// TwinCAT 3 PLC project Untitled1
// ProgramVersion: 3.1.4026.14
// libraries:
//   Tc2_EtherCAT, * (Beckhoff Automation GmbH)
//   Tc2_MC2, * (Beckhoff Automation GmbH)
//   Tc2_Standard, * (Beckhoff Automation GmbH)
//   Tc2_System, * (Beckhoff Automation GmbH)
//   Tc2_Utilities, * (Beckhoff Automation GmbH)
//   Tc3_Module, * (Beckhoff Automation GmbH)
// project tree:
//   DUTs/ ENUM_HardwareCheckState.TcDUT, ENUM_LinearActuatorState.TcDUT, ENUM_StepperMotorState.TcDUT, ST_AlarmEntry.TcDUT, ST_LinearActuator.TcDUT, ST_Alarm.TcDUT, ST_LinearActuatorCommand.TcDUT, ST_LinearTable.TcDUT, ST_LookupEntry.TcDUT, ST_StepperMotorCommand.TcDUT, ST_SystemAlarmStatus.TcDUT, ST_ZoneAlarmStatus.TcDUT
//   GVLs/ GVL_Alarms.TcGVL, GVL.TcGVL, GVL_CellPositionSensors.TcGVL, GVL_Steppers.TcGVL, GVL_LinearActuatorDriveControls.TcGVL, GVL_LinearActuatorProxSensors.TcGVL, GVL_LinearActuators.TcGVL, GVL_LinearActuatorRelays.TcGVL, GVL_Process.TcGVL, GVL_StepperPositions.TcGVL
//   / Main_Task.TcTTO
//   POUs/FunctionBlocks/ FB_AlarmStatusManager.TcPOU, FB_LinearActuator.TcPOU, FB_StepperMotor.TcPOU
//   POUs/Helper/ F_IssueActuatorCommand.TcPOU, F_GetLinearCommandMember.TcPOU, F_GetLinearCommandValue.TcPOU, F_GetStepperCommandMember.TcPOU, F_GetStepperCommandValue.TcPOU, F_GetStepperAlarmCondition.TcPOU, F_ValidateCommand.TcPOU, F_GetLinearActuatorAlarmCondition.TcPOU, F_GetMC2ErrorDescription.TcPOU
//   POUs/Programs/ PRG_AlarmHandler.TcPOU, PRG_CommandHandler.TcPOU, PRG_Cycle.TcPOU
// real-time tasks:
//   TASK Main_Task: cycle T#10ms, priority 1, ADS port 351
// motion (NC):
//   TASK NC-Task 1 SAF: cycle T#2ms, priority 4, ADS port 501
//   TASK NC-Task 1 SVB: cycle T#10ms, priority 12, ADS port 511
//   AXIS Stepper1 (id 1)
//     Dynamic: Acceleration=100, Deceleration=100, Jerk=66.6667
//     Velo: Maximum=150
//     OtherSettings: AllowMotionCmdToSlave=true
//     encoder EncType=19
//       EncPara: ScaleFactorNumerator=0.000115, MaxCount=#xffffffff
//         Inc: RefSoftSyncMask=#x0000ffff
//     drive DrvType=16
//       DrvPara: MaxCount=#xffffffff, DriveControlDWord=#x00020100
//         Analog: TorqueSetpointScale=10, ScaleFactorActTorque=0.1
//         TimeComp: TaskDelayCycles=1
//     controller CtrType=1
//       CtrPara: PriorControlFactor=1
//         Observer: BandWidth=20
//   AXIS Stepper2 (id 2)
//     Dynamic: Acceleration=99.9997, Deceleration=99.9997, Jerk=66.6667
//     Velo: Maximum=150
//     OtherSettings: AllowMotionCmdToSlave=true
//     encoder EncType=19
//       EncPara: MaxCount=#xffffffff
//         Inc: RefSoftSyncMask=#x0000ffff
//     drive DrvType=16
//       DrvPara: MaxCount=#xffffffff, DriveControlDWord=#x00020100
//         Analog: TorqueSetpointScale=10, ScaleFactorActTorque=0.1
//         TimeComp: TaskDelayCycles=1
//     controller CtrType=1
//       CtrPara: PriorControlFactor=1
//         Observer: BandWidth=20
//   AXIS Stepper3 (id 3)
//     Dynamic: Acceleration=100, Deceleration=100, Jerk=66.6667
//     Velo: Maximum=150
//     OtherSettings: AllowMotionCmdToSlave=true
//     encoder EncType=19
//       EncPara: MaxCount=#xffffffff
//         Inc: RefSoftSyncMask=#x0000ffff
//     drive DrvType=16
//       DrvPara: MaxCount=#xffffffff, DriveControlDWord=#x00020100
//         Analog: TorqueSetpointScale=10, ScaleFactorActTorque=0.1
//         TimeComp: TaskDelayCycles=1
//     controller CtrType=1
//       CtrPara: PriorControlFactor=1
//         Observer: BandWidth=20
//   AXIS Stepper4 (id 4)
//     Dynamic: Acceleration=100, Deceleration=100, Jerk=66.6667
//     Velo: Maximum=150
//     OtherSettings: AllowMotionCmdToSlave=true
//     encoder EncType=19
//       EncPara: MaxCount=#xffffffff
//         Inc: RefSoftSyncMask=#x0000ffff
//     drive DrvType=16
//       DrvPara: MaxCount=#xffffffff, DriveControlDWord=#x00020100
//         Analog: TorqueSetpointScale=10, ScaleFactorActTorque=0.1
//         TimeComp: TaskDelayCycles=1
//     controller CtrType=1
//       CtrPara: PriorControlFactor=1
//         Observer: BandWidth=20
// I/O:
//   DEVICE Périphérique 2 (EtherCAT) (disabled), AmsNetId 192.168.0.14.3.1
//     Terme 11 (EK1100) [EK1100 EtherCAT Coupler (2A E-Bus)]
//       Drive Stepper1 (EL7047) [EL7047 1Ch. Stepper motor output stage (50V, 5A)]
//       Drive Stepper2 (EL7047) [EL7047 1Ch. Stepper motor output stage (50V, 5A)]
//       Drive Stepper3 (EL7047) [EL7047 1Ch. Stepper motor output stage (50V, 5A)]
//       Drive Stepper4 (El7047) [EL7047 1Ch. Stepper motor output stage (50V, 5A)]
//   DEVICE Device 4 (EtherCAT) (disabled), AmsNetId 192.168.0.14.5.1
//     ECAT E-Bus (EK1200) [EK1200-5000 EtherCAT Power supply (2A E-Bus)]
//       Carte DO #1 (EL2809) [EL2809 16Ch. Dig. Output 24V, 0.5A]
//       Carte DO #2 (EL2809) [EL2809 16Ch. Dig. Output 24V, 0.5A]
//       Carte DO #3 (EL2809) [EL2809 16Ch. Dig. Output 24V, 0.5A]
//       Drive Stepper Rail1/2 (EL7062) [EL7062-0000 2Ch. Stepper motor output stage (48V, 3A)]
//       Drive Stepper Rail3/4 (EL7062) [EL7062-0000 2Ch. Stepper motor output stage (48V, 3A)]
//       E-Bus (EL9410) [EL9410 E-Bus Power Supplier  (Diagnostics)]
//       Carte DI #1 (EL1409) [EL1409 16Ch. Dig. Input 24V, 3ms]
//       Carte DI #2 (EL1409) [EL1409 16Ch. Dig. Input 24V, 3ms]
//       Carte DI #3 (EL1409) [EL1409 16Ch. Dig. Input 24V, 3ms]
//       Term 10 (EL4074) [EL4074 4K. Ana. Ausgang, +/-10V, +/-20mA, 16 Bit]
//       Term 8 (EL3078) [EL3078 8K. Ana. Eingang  +/-10V, +/-20mA]
//       Term 9 (EL3078) [EL3078 8K. Ana. Eingang  +/-10V, +/-20mA]
//       Carte Temperature Sensors #1 (EL3208-0010) [EL3208-0010 8Ch. Ana. Input PT1000 (RTD)]
//       Carte Temperature Sensors #2 (EL3208-0010) [EL3208-0010 8Ch. Ana. Input PT1000 (RTD)]
//       Carte Temperature Sensors #3 (EL3208-0010) [EL3208-0010 8Ch. Ana. Input PT1000 (RTD)]
//       End Terminal (EL9011) [EL9011 End Terminal]
// variable links:
//   NC-Task 1 SAF/Axes/Stepper1 <-> Device 4 (EtherCAT)/ECAT E-Bus (EK1200)/Drive Stepper Rail1/2 (EL7062)
//     Drive/Inputs/In/nDataIn1 <-> DRV Following error actual value Channel 1/Following error actual value
//     Drive/Inputs/In/nDcOutputTime <-> InfoData/DcOutputShift
//     Drive/Inputs/In/nState1 <-> DRV Statusword Channel 1/Statusword
//     Drive/Inputs/In/nState2 <-> DRV Statusword Channel 1/Statusword @bit 8
//     Drive/Inputs/In/nState4 @bit 1 <-> WcState/InputToggle
//     Drive/Inputs/In/nState4 <-> WcState/WcState
//     Drive/Outputs/Out/nCtrl1 <-> DRV Controlword Channel 1/Controlword
//     Drive/Outputs/Out/nCtrl2 <-> DRV Controlword Channel 1/Controlword @bit 8
//     Drive/Outputs/Out/nDataOut1 <-> DRV Target position Channel 1/Target position
//     Enc/Inputs/In/nDataIn1 <-> FB Position Channel 1/Position
//     Enc/Inputs/In/nDcInputTime <-> InfoData/DcInputShift
//     Enc/Inputs/In/nState4 @bit 1 <-> WcState/InputToggle
//     Enc/Inputs/In/nState4 <-> WcState/WcState
//   NC-Task 1 SAF/Axes/Stepper2 <-> Device 4 (EtherCAT)/ECAT E-Bus (EK1200)/Drive Stepper Rail1/2 (EL7062)
//     Drive/Inputs/In/nDataIn1 <-> DRV Following error actual value Channel 2/Following error actual value
//     Drive/Inputs/In/nDcOutputTime <-> InfoData/DcOutputShift
//     Drive/Inputs/In/nState1 <-> DRV Statusword Channel 2/Statusword
//     Drive/Inputs/In/nState2 <-> DRV Statusword Channel 2/Statusword @bit 8
//     Drive/Inputs/In/nState4 @bit 1 <-> WcState/InputToggle
//     Drive/Inputs/In/nState4 <-> WcState/WcState
//     Drive/Outputs/Out/nCtrl1 <-> DRV Controlword Channel 2/Controlword
//     Drive/Outputs/Out/nCtrl2 <-> DRV Controlword Channel 2/Controlword @bit 8
//     Drive/Outputs/Out/nDataOut1 <-> DRV Target position Channel 2/Target position
//     Enc/Inputs/In/nDataIn1 <-> FB Position Channel 2/Position
//     Enc/Inputs/In/nDcInputTime <-> InfoData/DcInputShift
//     Enc/Inputs/In/nState4 @bit 1 <-> WcState/InputToggle
//     Enc/Inputs/In/nState4 <-> WcState/WcState
//   NC-Task 1 SAF/Axes/Stepper3 <-> Device 4 (EtherCAT)/ECAT E-Bus (EK1200)/Drive Stepper Rail3/4 (EL7062)
//     Drive/Inputs/In/nDataIn1 <-> DRV Following error actual value Channel 1/Following error actual value
//     Drive/Inputs/In/nDcOutputTime <-> InfoData/DcOutputShift
//     Drive/Inputs/In/nState1 <-> DRV Statusword Channel 1/Statusword
//     Drive/Inputs/In/nState2 <-> DRV Statusword Channel 1/Statusword @bit 8
//     Drive/Inputs/In/nState4 @bit 1 <-> WcState/InputToggle
//     Drive/Inputs/In/nState4 <-> WcState/WcState
//     Drive/Outputs/Out/nCtrl1 <-> DRV Controlword Channel 1/Controlword
//     Drive/Outputs/Out/nCtrl2 <-> DRV Controlword Channel 1/Controlword @bit 8
//     Drive/Outputs/Out/nDataOut1 <-> DRV Target position Channel 1/Target position
//     Enc/Inputs/In/nDataIn1 <-> FB Position Channel 1/Position
//     Enc/Inputs/In/nDcInputTime <-> InfoData/DcInputShift
//     Enc/Inputs/In/nState4 @bit 1 <-> WcState/InputToggle
//     Enc/Inputs/In/nState4 <-> WcState/WcState
//   NC-Task 1 SAF/Axes/Stepper4 <-> Device 4 (EtherCAT)/ECAT E-Bus (EK1200)/Drive Stepper Rail3/4 (EL7062)
//     Drive/Inputs/In/nDataIn1 <-> DRV Following error actual value Channel 2/Following error actual value
//     Drive/Inputs/In/nDcOutputTime <-> InfoData/DcOutputShift
//     Drive/Inputs/In/nState1 <-> DRV Statusword Channel 2/Statusword
//     Drive/Inputs/In/nState2 <-> DRV Statusword Channel 2/Statusword @bit 8
//     Drive/Inputs/In/nState4 @bit 1 <-> WcState/InputToggle
//     Drive/Inputs/In/nState4 <-> WcState/WcState
//     Drive/Outputs/Out/nCtrl1 <-> DRV Controlword Channel 2/Controlword
//     Drive/Outputs/Out/nCtrl2 <-> DRV Controlword Channel 2/Controlword @bit 8
//     Drive/Outputs/Out/nDataOut1 <-> DRV Target position Channel 2/Target position
//     Enc/Inputs/In/nDataIn1 <-> FB Position Channel 2/Position
//     Enc/Inputs/In/nDcInputTime <-> InfoData/DcInputShift
//     Enc/Inputs/In/nState4 @bit 1 <-> WcState/InputToggle
//     Enc/Inputs/In/nState4 <-> WcState/WcState
//   Untitled1/Untitled1 Instance <-> Device 4 (EtherCAT)/ECAT E-Bus (EK1200)/Carte DI #1 (EL1409)
//     Main_Task Inputs/GVL_CellPositionSensors.Cell_Pos{1..6} <-> DIP Inputs/Cell Position {1..6}  (6 links)
//     Main_Task Inputs/GVL_LinearActuatorProxSensors.Tri{1..4}_Prox_In <-> DIP Inputs/Triangle Rétractable Chariot{1..4} Prox In  (4 links)
//     Main_Task Inputs/GVL_LinearActuatorProxSensors.Tri{1..4}_Prox_Out <-> DIP Inputs/Triangle Rétractable Chariot{1..4} Prox Out  (4 links)
//   Untitled1/Untitled1 Instance <-> Device 4 (EtherCAT)/ECAT E-Bus (EK1200)/Carte DI #2 (EL1409)
//     Main_Task Inputs/GVL_LinearActuatorProxSensors.Gui1_Prox_In_Slow <-> DIP Inputs/Gui1 Prox In Slow
//     Main_Task Inputs/GVL_LinearActuatorProxSensors.Gui2_Prox_In_Slow <-> DIP Inputs/Gui2 Prox In Slow
//     Main_Task Inputs/GVL_LinearActuatorProxSensors.Gui1_Prox_Out <-> DIP Inputs/Gui1 Prox Out
//     Main_Task Inputs/GVL_LinearActuatorProxSensors.Gui2_Prox_Out <-> DIP Inputs/Gui2 Prox Out
//     Main_Task Inputs/GVL_LinearActuatorProxSensors.Gui1_Prox_Out_Slow <-> DIP Inputs/Gui1 Prox Out Slow
//     Main_Task Inputs/GVL_LinearActuatorProxSensors.Gui2_Prox_Out_Slow <-> DIP Inputs/Gui2 Prox Out Slow
//     Main_Task Inputs/GVL_Steppers.Rail1_Prox <-> DIP Inputs/Prox Homing Rail1
//     Main_Task Inputs/GVL_Steppers.Rail2_Prox <-> DIP Inputs/Prox Homing Rail2
//   Untitled1/Untitled1 Instance <-> Device 4 (EtherCAT)/ECAT E-Bus (EK1200)/Carte DI #3 (EL1409)
//     Main_Task Inputs/GVL.PLC_Fan_Steppers <-> DIP Inputs/Fan Stepper Status
//     Main_Task Inputs/GVL.ResetSafety <-> DIP Inputs/Reset Safety
//     Main_Task Inputs/GVL.SafetyRelayStatus <-> DIP Inputs/Safety Relay Status
//     Main_Task Inputs/GVL.StartCycle <-> DIP Inputs/Start Cycle
//     Main_Task Inputs/GVL.StopCycle <-> DIP Inputs/Stop Cycle
//     Main_Task Inputs/GVL_LinearActuatorDriveControls.Cmp1_Mot_Fault <-> DIP Inputs/Cmp1 Fault
//     Main_Task Inputs/GVL_LinearActuatorDriveControls.Cmp2_Mot_Fault <-> DIP Inputs/Cmp2 Fault
//     Main_Task Inputs/GVL_LinearActuatorDriveControls.Gui1_Mot_Fault <-> DIP Inputs/Gui1 Fault
//     Main_Task Inputs/GVL_LinearActuatorDriveControls.Gui2_Mot_Fault <-> DIP Inputs/Gui2 Fault
//     Main_Task Inputs/GVL_LinearActuatorProxSensors.Piv1_Prox_In <-> DIP Inputs/Piv1 Prox In
//     Main_Task Inputs/GVL_LinearActuatorProxSensors.Piv1_Prox_Out <-> DIP Inputs/Piv1 Prox Out
//     Main_Task Inputs/GVL_Steppers.Rail3_Prox <-> DIP Inputs/Prox Homing Rail3
//     Main_Task Inputs/GVL_Steppers.Rail4_Prox <-> DIP Inputs/Prox Homing Rail4
//   Untitled1/Untitled1 Instance <-> Device 4 (EtherCAT)/ECAT E-Bus (EK1200)/Carte DO #2 (EL2809)
//     Main_Task Outputs/GVL_LinearActuatorRelays.Piv1_Mot_Bw <-> Channel 13/Piv1 Backward
//     Main_Task Outputs/GVL_LinearActuatorRelays.Piv1_Mot_Fw <-> Channel 5/Piv1 Forward
//     Main_Task Outputs/GVL_LinearActuatorRelays.Tri1_Mot_Bw <-> Channel 1/Tri1 Pop-Up Forward
//     Main_Task Outputs/GVL_LinearActuatorRelays.Tri1_Mot_Fw <-> Channel 9/Tri1 Pop-Up Backward
//     Main_Task Outputs/GVL_LinearActuatorRelays.Tri2_Mot_Bw <-> Channel 11/Tri2 Pop-Up Backward
//     Main_Task Outputs/GVL_LinearActuatorRelays.Tri3_Mot_Bw <-> Channel 12/Tri3 Pop-Up Backward
//     Main_Task Outputs/GVL_LinearActuatorRelays.Tri4_Mot_Bw <-> Channel 10/Tri4 Pop-Up Backward
//     Main_Task Outputs/GVL_LinearActuatorRelays.Tri2_Mot_Fw <-> Channel 3/Tri2 Pop-Up Forward
//     Main_Task Outputs/GVL_LinearActuatorRelays.Tri3_Mot_Fw <-> Channel 4/Tri3 Pop-Up Forward
//     Main_Task Outputs/GVL_LinearActuatorRelays.Tri4_Mot_Fw <-> Channel 2/Tri4 Forward
//   Untitled1/Untitled1 Instance <-> Device 4 (EtherCAT)/ECAT E-Bus (EK1200)/Carte DO #3 (EL2809)
//     Main_Task Outputs/GVL_LinearActuatorDriveControls.Cmp1_Mot_Speed2 <-> Channel 4/Cmp1 Speed2
//     Main_Task Outputs/GVL_LinearActuatorDriveControls.Cmp2_Mot_Speed2 <-> Channel 16/Cmp2 Speed2
//     Main_Task Outputs/GVL_LinearActuatorDriveControls.Cmp1_Mot_Stop <-> Channel 3/Cmp1 Stop
//     Main_Task Outputs/GVL_LinearActuatorDriveControls.Cmp2_Mot_Stop <-> Channel 15/Cmp2 Stop
//     Main_Task Outputs/GVL_LinearActuatorDriveControls.Gui1_Mot_Speed2 <-> Channel 8/Gui1 Speed2
//     Main_Task Outputs/GVL_LinearActuatorDriveControls.Gui2_Mot_Speed2 <-> Channel 12/Gui2 Speed2
//     Main_Task Outputs/GVL_LinearActuatorDriveControls.Gui1_Mot_Stop <-> Channel 7/Gui1 Stop
//     Main_Task Outputs/GVL_LinearActuatorDriveControls.Gui2_Mot_Stop <-> Channel 11/Gui2 Stop
//     Main_Task Outputs/GVL_LinearActuatorRelays.Cmp1_Mot_Bw <-> Channel 1/Cmp1 Backward
//     Main_Task Outputs/GVL_LinearActuatorRelays.Cmp2_Mot_Bw <-> Channel 13/Cmp2 Backward
//     Main_Task Outputs/GVL_LinearActuatorRelays.Cmp1_Mot_Fw <-> Channel 2/Cmp1 Forward
//     Main_Task Outputs/GVL_LinearActuatorRelays.Cmp2_Mot_Fw <-> Channel 14/Cmp2 Forward
//     Main_Task Outputs/GVL_LinearActuatorRelays.Gui1_Mot_Bw <-> Channel 5/Gui1 Backward
//     Main_Task Outputs/GVL_LinearActuatorRelays.Gui2_Mot_Bw <-> Channel 9/Gui2 Backward
//     Main_Task Outputs/GVL_LinearActuatorRelays.Gui1_Mot_Fw <-> Channel 6/Gui1 Forward
//     Main_Task Outputs/GVL_LinearActuatorRelays.Gui2_Mot_Fw <-> Channel 10/Gui2 Forward
//   Untitled1/Untitled1 Instance <-> NC-Task 1 SAF/Axes/Stepper1
//     Main_Task Inputs/GVL_Steppers.Rail1_Mot_Struct.object.NcToPlc <-> Outputs/ToPlc
//     Main_Task Outputs/GVL_Steppers.Rail1_Mot_Struct.object.PlcToNc <-> Inputs/FromPlc
//   Untitled1/Untitled1 Instance <-> NC-Task 1 SAF/Axes/Stepper2
//     Main_Task Inputs/GVL_Steppers.Rail2_Mot_Struct.object.NcToPlc <-> Outputs/ToPlc
//     Main_Task Outputs/GVL_Steppers.Rail2_Mot_Struct.object.PlcToNc <-> Inputs/FromPlc
//   Untitled1/Untitled1 Instance <-> NC-Task 1 SAF/Axes/Stepper3
//     Main_Task Inputs/GVL_Steppers.Rail3_Mot_Struct.object.NcToPlc <-> Outputs/ToPlc
//     Main_Task Outputs/GVL_Steppers.Rail3_Mot_Struct.object.PlcToNc <-> Inputs/FromPlc
//   Untitled1/Untitled1 Instance <-> NC-Task 1 SAF/Axes/Stepper4
//     Main_Task Inputs/GVL_Steppers.Rail4_Mot_Struct.object.NcToPlc <-> Outputs/ToPlc
//     Main_Task Outputs/GVL_Steppers.Rail4_Mot_Struct.object.PlcToNc <-> Inputs/FromPlc

CONFIGURATION Untitled1
    RESOURCE PLC ON TwinCAT3
        TASK Main_Task(INTERVAL := T#10ms, PRIORITY := 1);
        PROGRAM PRG_Cycle WITH Main_Task : PRG_Cycle;
        PROGRAM PRG_AlarmHandler WITH Main_Task : PRG_AlarmHandler;
        PROGRAM PRG_CommandHandler WITH Main_Task : PRG_CommandHandler;
    END_RESOURCE
END_CONFIGURATION

// ---- DUTs/ENUM_HardwareCheckState.TcDUT
TYPE ENUM_HardwareCheckState :
(
	HW_Start := 0,
	HW_Complete := 1,
	HW_Failed := 2
);
END_TYPE

// ---- DUTs/ENUM_LinearActuatorState.TcDUT
TYPE ENUM_LinearActuatorState :
(
    LAS_LinearActuator_Extending := 0,
    LAS_LinearActuator_Extended := 1,
    LAS_LinearActuator_Retracting := 2,
    LAS_LinearActuator_Retracted := 3,
    LAS_LinearActuator_Error := 4,
	LAS_LinearActuator_AtProx2 := 5,    
    LAS_LinearActuator_AtProx3 := 6,
	LAS_LinearActuator_Uninitialised := 7  
);
END_TYPE

// ---- DUTs/ENUM_StepperMotorState.TcDUT
TYPE ENUM_StepperMotorState :
(
	LAS_Stepper_Ready := 0,
    LAS_Stepper_Moving := 1,
    LAS_Stepper_Idle := 2,
    LAS_Stepper_Error := 3,
	LAS_Stepper_Homing := 4,
	LAS_Stepper_Hardware_Check := 5,
	LAS_Stepper_PowerError := 6
);
END_TYPE

// ---- DUTs/ST_AlarmEntry.TcDUT
TYPE ST_AlarmEntry :
STRUCT
    pAlarm : POINTER TO ST_Alarm;     
    sName : STRING(50);               
END_STRUCT
END_TYPE

// ---- DUTs/ST_LinearActuator.TcDUT
TYPE ST_LinearActuator :
STRUCT
    sName : STRING(50);
    bProxIn : POINTER TO BOOL;      
    bProxOut : POINTER TO BOOL;    
    bProx2 : POINTER TO BOOL;       
    bProx3 : POINTER TO BOOL;       
    bFwdDO   : POINTER TO BOOL;     
    bBckwDO  : POINTER TO BOOL;     
    bSpeedControlDO : POINTER TO BOOL; 
	bStopControlDO : POINTER TO BOOL;
    bFaultDI : POINTER TO BOOL;     
    tTimeout : TON;
END_STRUCT
END_TYPE

// ---- DUTs/ST_Alarm.TcDUT
TYPE ST_Alarm :
STRUCT
    bCondition      : BOOL;           
    nID             : UDINT;           
    nSeverity       : UINT;     
	sMessage        : STRING(255);        
END_STRUCT
END_TYPE

// ---- DUTs/ST_LinearActuatorCommand.TcDUT
TYPE ST_LinearActuatorCommand :
STRUCT
	bCommand : BOOL;
	nStatus : SINT;
END_STRUCT
END_TYPE

// ---- DUTs/ST_LinearTable.TcDUT
TYPE ST_LinearTable :
STRUCT
	object : AXIS_REF;
	bProx : POINTER TO BOOL;
	fReferencePos : LREAL;
	stHomingOptions : ST_HomingOptions;
END_STRUCT
END_TYPE

// ---- DUTs/ST_LookupEntry.TcDUT
TYPE ST_LookupEntry :
STRUCT
    nX : SINT;
    sY : STRING;
    sValue: POINTER TO FB_LinearActuator;
	sCommand: POINTER TO ST_LinearActuatorCommand;
END_STRUCT
END_TYPE

// ---- DUTs/ST_StepperMotorCommand.TcDUT
TYPE ST_StepperMotorCommand :
STRUCT
	bHoming : BOOL;
	nCommand : LREAL;
	fVelocity : LREAL;
	nPosition : LREAL;
	bHomed : BOOL;
END_STRUCT
END_TYPE

// ---- DUTs/ST_SystemAlarmStatus.TcDUT
TYPE ST_SystemAlarmStatus :
STRUCT
    bGlobalOkToRun : BOOL;                            
    bAllZonesOk : BOOL;                                
    aZoneStatus : ARRAY[1..5] OF ST_ZoneAlarmStatus;    
    bMaintenanceMode : BOOL;                          
END_STRUCT
END_TYPE

// ---- DUTs/ST_ZoneAlarmStatus.TcDUT
TYPE ST_ZoneAlarmStatus :
STRUCT
    bOkToRun : BOOL;           
    nHighestSeverity : UINT;   
END_STRUCT
END_TYPE

// ---- GVLs/GVL_Alarms.TcGVL
VAR_GLOBAL
	
	// ================================================================
    // RAIL 1
    // ================================================================
	R1_Sensor_UnknownPosition : ST_Alarm := (
		nID := 1001,
		nSeverity := 3);
	
	R1_Sensor_MotionTimedOut : ST_Alarm := (
		nID := 1002,
		nSeverity := 3);
	
	R1_Chariot_UnknownPosition : ST_Alarm := (
		nID := 1003,
		nSeverity := 3);
	
	R1_Chariot_MotionTimedOut : ST_Alarm := (
		nID := 1004,
		nSeverity := 3);
	
	R1_Compressor_UnknownPosition : ST_Alarm := (
		nID := 1005,
		nSeverity := 3);
	
	R1_Compressor_MotionTimedOut : ST_Alarm := (
		nID := 1006,
		nSeverity := 3);
	
	R1_Stepper_Motion_Failed : ST_Alarm := (
		sMessage := '',
		nID := 1007,
		nSeverity := 3);
	
	R1_Stepper_Homing_Failed : ST_Alarm := (
		sMessage := '',
		nID := 1008,
		nSeverity := 3);
	
	R1_Stepper_Motion_Interrupted : ST_Alarm := (
		sMessage := '',
		nID := 1010,
		nSeverity := 3);
	
	R1_Stepper_PowerUp_Failed : ST_Alarm := (
		sMessage := '',
		nID := 1011,
		nSeverity := 3);
	
	R1_Stepper_Reset_Failed : ST_Alarm := (
		sMessage := '',
		nID := 1012,
		nSeverity := 3);
	
	R1_Stepper_Stop_Failed : ST_Alarm := (
		sMessage := '',
		nID := 1013,
		nSeverity := 3);
	
	R1_Stepper_UnableToReadPosition : ST_Alarm := (
		sMessage := '',
		nID := 1014,
		nSeverity := 3);
	
	R1_Compressor_DriveFaulted : ST_Alarm := (
		nID := 1015,
		nSeverity := 5);
	
	
	// ================================================================
    // RAIL 2
    // ================================================================
	R2_Stepper_PowerUp_Failed : ST_Alarm := (
		sMessage := '',
		nID := 2001,
		nSeverity := 3);
	
	R2_Stepper_Homing_Failed : ST_Alarm := (
		sMessage := '',
		nID := 2002,
		nSeverity := 3);
	
	R2_Stepper_Motion_Failed : ST_Alarm := (
		sMessage := '',
		nID := 2004,
		nSeverity := 3);
	
	R2_Stepper_Motion_Interrupted : ST_Alarm := (
		sMessage := '',
		nID := 2005,
		nSeverity := 3);
	
	R2_Stepper_Reset_Failed : ST_Alarm := (
		sMessage := '',
		nID := 2006,
		nSeverity := 3);
		
	R2_Chariot_UnknownPosition : ST_Alarm := (
		nID := 2007,
		nSeverity := 3);
	
	R2_Chariot_MotionTimedOut : ST_Alarm := (
		nID := 2008,
		nSeverity := 3);
	
	R2_Stepper_Stop_Failed : ST_Alarm := (
		sMessage := '',
		nID := 2009,
		nSeverity := 3);
	
	R2_Stepper_UnableToReadPosition : ST_Alarm := (
		sMessage := '',
		nID := 2010,
		nSeverity := 3);
	
	
	// ================================================================
    // RAIL 3
    // ================================================================
	R3_Compressor_UnknownPosition : ST_Alarm := (
		nID := 3001,
		nSeverity := 3);
	
	R3_Compressor_MotionTimedOut : ST_Alarm := (
		nID := 3002,
		nSeverity := 3);
	
	R3_HeatExCoupola_UnknownState : ST_Alarm := (
		nID := 3003,
		nSeverity := 3);
	
	R3_HeatExCoupola_MotionTimedOut : ST_Alarm := (
		nID := 3004,
		nSeverity := 3);
	
	R3_RegenCoupola_UnknownPosition : ST_Alarm := (
		nID := 3005,
		nSeverity := 3);
	
	R3_RegenCoupola_MotionTimedOut : ST_Alarm := (
		nID := 3006,
		nSeverity := 3);
	
	R3_Chariot_UnknownPosition : ST_Alarm := (
		nID := 3007,
		nSeverity := 3);
	
	R3_Chariot_MotionTimedOut : ST_Alarm := (
		nID := 3008,
		nSeverity := 3);
		
	R3_Stepper_PowerUp_Failed : ST_Alarm := (
		sMessage := '',
		nID := 3009,
		nSeverity := 3);
	
	R3_Stepper_Homing_Failed : ST_Alarm := (
		sMessage := '',
		nID := 3010,
		nSeverity := 3);
	
	R3_Stepper_Motion_Failed : ST_Alarm := (
		sMessage := '',
		nID := 3012,
		nSeverity := 3);
	
	R3_Stepper_Motion_Interrupted : ST_Alarm := (
		sMessage := '',
		nID := 3013,
		nSeverity := 3);
	
	R3_Stepper_Reset_Failed : ST_Alarm := (
		sMessage := '',
		nID := 3014,
		nSeverity := 3);
	
	R3_Stepper_Stop_Failed : ST_Alarm := (
		sMessage := '',
		nID := 3015,
		nSeverity := 3);
	
	R3_HeatExCoupola_DriveFaulted : ST_Alarm := (
		nID := 3016,
		nSeverity := 5);
	
	R3_RegenCoupola_DriveFaulted : ST_Alarm := (
		nID := 3017,
		nSeverity := 5);
	
	R3_Stepper_UnableToReadPosition : ST_Alarm := (
		sMessage := '',
		nID := 3018,
		nSeverity := 3);
	
	R3_Compressor_DriveFaulted : ST_Alarm := (
		nID := 3019,
		nSeverity := 5);
	
	// ================================================================
    // RAIL 4
    // ================================================================
	R4_Stepper_PowerUp_Failed : ST_Alarm := (
		sMessage := '',
		nID := 4001,
		nSeverity := 3);
	
	R4_Stepper_Homing_Failed : ST_Alarm := (
		sMessage := '',
		nID := 4002,
		nSeverity := 3);
	
	R4_Stepper_Motion_Failed : ST_Alarm := (
		sMessage := '',
		nID := 4004,
		nSeverity := 3);
	
	R4_Stepper_Motion_Interrupted : ST_Alarm := (
		sMessage := '',
		nID := 4005,
		nSeverity := 3);
	
	R4_Stepper_Reset_Failed : ST_Alarm := (
		sMessage := '',
		nID := 4006,
		nSeverity := 3);
	
	R4_Chariot_UnknownPosition : ST_Alarm := (
		nID := 4007,
		nSeverity := 3);
	
	R4_Chariot_MotionTimedOut : ST_Alarm := (
		nID := 4008,
		nSeverity := 3);
	
	R4_Stepper_Stop_Failed : ST_Alarm := (
		sMessage := '',
		nID := 4009,
		nSeverity := 3);
	
	R4_Stepper_UnableToReadPosition : ST_Alarm := (
		sMessage := '',
		nID := 4010,
		nSeverity := 3);
	
	
	// ================================================================
    // GLOBAL SECURITY (ZONE 5)
    // ================================================================
	SafetyRelay : ST_Alarm := (
		nID := 9001,
		nSeverity := 5);
	
	bCriticalAlarm : BOOL;
END_VAR

// ---- GVLs/GVL.TcGVL
{attribute 'global_init_slot' := '1'}
VAR_GLOBAL
	
	StartCycle AT %I*: BOOL;
	StartCycle_HMI : BOOL;
	StopCycle AT %I*: BOOL;
	StopCycle_HMI : BOOL;
	ResetSafety AT %I*: BOOL;

    RTrigStart : R_TRIG;
    RTrigStop  : R_TRIG;

    bStartCycleMem : BOOL;  
    bStopCycleMem  : BOOL;  
	
	SafetyRelayStatus AT %I*: BOOL;
	
	gSystemAlarmStatus : ST_SystemAlarmStatus;
	
	PLC_Fan_Steppers AT %I*: BOOL;
	
	CONTROL : BOOL := FALSE;
	
	Result          : INT := 0;
	
	sRequestedActuator : STRING := '';
	bIsPoweredUp     : ARRAY[1..4] OF BOOL;
	
	aLookupTable : ARRAY[1..100] OF ST_LookupEntry := [
		(nX := 1, sY := 'Chariot', sValue := ADR(Tri1_Mot_FB), sCommand := ADR(Tri1_Mot_Cmd)),
		(nX := 1, sY := 'Compressor', sValue := ADR(Cmp1_Mot_FB), sCommand := ADR(Cmp1_Mot_Cmd)),
		(nX := 1, sY := 'Sensor', sValue := ADR(Piv1_Mot_FB), sCommand := ADR(Piv1_Mot_Cmd)),
		(nX := 2, sY := 'Chariot', sValue := ADR(Tri2_Mot_FB), sCommand := ADR(Tri2_Mot_Cmd)),
		(nX := 3, sY := 'HeatExCoupola', sValue := ADR(Gui1_Mot_FB), sCommand := ADR(Gui1_Mot_Cmd)),
		(nX := 3, sY := 'RegenCoupola', sValue := ADR(Gui2_Mot_FB), sCommand := ADR(Gui2_Mot_Cmd)),
		(nX := 3, sY := 'Chariot', sValue := ADR(Tri3_Mot_FB), sCommand := ADR(Tri3_Mot_Cmd)),
		(nX := 3, sY := 'Compressor', sValue := ADR(Cmp2_Mot_FB), sCommand := ADR(Cmp2_Mot_Cmd)),
		(nX := 4, sY := 'Chariot', sValue := ADR(Tri4_Mot_FB), sCommand := ADR(Tri4_Mot_Cmd)),
		(nX := 1, sY := 'Home', sValue := ADR(Rail1_Mot_FB), sCommand := ADR(Rail1_Mot_Cmd)),
		(nX := 1, sY := 'Motor', sValue := ADR(Rail1_Mot_FB), sCommand := ADR(Rail1_Mot_Cmd)),
		(nX := 2, sY := 'Home', sValue := ADR(Rail2_Mot_FB), sCommand := ADR(Rail2_Mot_Cmd)),
		(nX := 2, sY := 'Motor', sValue := ADR(Rail2_Mot_FB), sCommand := ADR(Rail2_Mot_Cmd)),
		(nX := 3, sY := 'Home', sValue := ADR(Rail3_Mot_FB), sCommand := ADR(Rail3_Mot_Cmd)),
		(nX := 3, sY := 'Motor', sValue := ADR(Rail3_Mot_FB), sCommand := ADR(Rail3_Mot_Cmd)),
		(nX := 4, sY := 'Motor', sValue := ADR(Rail4_Mot_FB), sCommand := ADR(Rail4_Mot_Cmd)),
		(nX := 4, sY := 'Motor', sValue := ADR(Rail4_Mot_FB), sCommand := ADR(Rail4_Mot_Cmd))
	];
    nEntryCount : INT := 17; 
END_VAR

// ---- GVLs/GVL_CellPositionSensors.TcGVL
VAR_GLOBAL
	Cell_Pos1 AT %I* : BOOL;
	Cell_Pos2 AT %I* : BOOL;
	Cell_Pos3 AT %I* : BOOL;
	
	Cell_Pos4 AT %I* : BOOL;
	Cell_Pos5 AT %I* : BOOL;
	Cell_Pos6 AT %I* : BOOL;
END_VAR

// ---- GVLs/GVL_Steppers.TcGVL
VAR_GLOBAL
	Rail1_Mot_Ref : AXIS_REF;
	Rail2_Mot_Ref : AXIS_REF;
	Rail3_Mot_Ref : AXIS_REF;
	Rail4_Mot_Ref : AXIS_REF;
	
	Rail1_Prox AT %I* : BOOL;
	Rail2_Prox AT %I* : BOOL;
	Rail3_Prox AT %I* : BOOL;
	Rail4_Prox AT %I* : BOOL;
	
	Mot_LoadedVel : LREAL := 50;
	Mot_HomingVel : LREAL := 50;
	Mot_UnloadedVel : LREAL := 250;
	
	Rail1_Mot_Struct : ST_LinearTable := (
		object := Rail1_Mot_Ref,
		bProx := ADR(Rail1_Prox),
		fReferencePos := 18.1,
		stHomingOptions := (SearchVelocity := Mot_HomingVel, SearchDirection := MC_Negative_Direction, ReferenceMode := ENCODERREFERENCEMODE_PLCCAM, SyncDirection := MC_Positive_Direction)
		);
	
	Rail2_Mot_Struct : ST_LinearTable := (
		object := Rail2_Mot_Ref,
		bProx := ADR(Rail2_Prox),
		fReferencePos := 10.0,
		stHomingOptions := (SearchVelocity := Mot_HomingVel, SearchDirection := MC_Negative_Direction, ReferenceMode := ENCODERREFERENCEMODE_PLCCAM, SyncDirection := MC_Positive_Direction)
		);
	
	Rail3_Mot_Struct : ST_LinearTable := (
		object := Rail3_Mot_Ref,
		bProx := ADR(Rail3_Prox),
		fReferencePos := 10.0,
		stHomingOptions := (SearchVelocity := Mot_HomingVel, SearchDirection := MC_Negative_Direction, ReferenceMode := ENCODERREFERENCEMODE_PLCCAM, SyncDirection := MC_Positive_Direction)
		);
	
	Rail4_Mot_Struct : ST_LinearTable := (
		object := Rail4_Mot_Ref,
		bProx := ADR(Rail4_Prox),
		fReferencePos := 10.0,
		stHomingOptions := (SearchVelocity := Mot_HomingVel, SearchDirection := MC_Negative_Direction, ReferenceMode := ENCODERREFERENCEMODE_PLCCAM, SyncDirection := MC_Positive_Direction)
		);
	
	Rail1_Mot_FB : FB_StepperMotor(init_axis := ADR(Rail1_Mot_Struct.object), init_prox := Rail1_Mot_Struct.bProx, init_refpos := ADR(Rail1_Mot_Struct.fReferencePos), init_homingoptions := ADR(Rail1_Mot_Struct.stHomingOptions));
    Rail2_Mot_FB : FB_StepperMotor(init_axis := ADR(Rail2_Mot_Struct.object), init_prox := Rail2_Mot_Struct.bProx, init_refpos := ADR(Rail2_Mot_Struct.fReferencePos), init_homingoptions := ADR(Rail2_Mot_Struct.stHomingOptions));
    Rail3_Mot_FB : FB_StepperMotor(init_axis := ADR(Rail3_Mot_Struct.object), init_prox := Rail3_Mot_Struct.bProx, init_refpos := ADR(Rail3_Mot_Struct.fReferencePos), init_homingoptions := ADR(Rail3_Mot_Struct.stHomingOptions));
    Rail4_Mot_FB : FB_StepperMotor(init_axis := ADR(Rail4_Mot_Struct.object), init_prox := Rail4_Mot_Struct.bProx, init_refpos := ADR(Rail4_Mot_Struct.fReferencePos), init_homingoptions := ADR(Rail4_Mot_Struct.stHomingOptions));

	Rail1_Mot_Cmd : ST_StepperMotorCommand := (
		bHoming := FALSE,
		nCommand := 0,
		nPosition := -1,
		bHomed := FALSE)
	;
	Rail2_Mot_Cmd : ST_StepperMotorCommand := (
		bHoming := FALSE,
		nCommand := 0,
		nPosition := -1,
		bHomed := FALSE)
	;
	Rail3_Mot_Cmd : ST_StepperMotorCommand := (
		bHoming := FALSE,
		nCommand := 0,
		nPosition := -1,
		bHomed := FALSE)
	;
	Rail4_Mot_Cmd : ST_StepperMotorCommand := (
		bHoming := FALSE,
		nCommand := 0,
		nPosition := -1,
		bHomed := FALSE)
	;
END_VAR

// ---- GVLs/GVL_LinearActuatorDriveControls.TcGVL
VAR_GLOBAL
	Gui1_Mot_Speed2 AT %Q* : BOOL;
	Gui1_Mot_Stop AT %Q* : BOOL;
	Gui1_Mot_Fault AT %I* : BOOL;
	
	Gui2_Mot_Speed2 AT %Q* : BOOL;
	Gui2_Mot_Stop AT %Q* : BOOL;
	Gui2_Mot_Fault AT %I* : BOOL;
	
	Cmp1_Mot_Speed2 AT %Q* : BOOL;
	Cmp1_Mot_Stop AT %Q* : BOOL;
	Cmp1_Mot_Fault AT %I* : BOOL;
	
	Cmp2_Mot_Speed2 AT %Q* : BOOL;
	Cmp2_Mot_Stop AT %Q* : BOOL;
	Cmp2_Mot_Fault AT %I* : BOOL;
END_VAR

// ---- GVLs/GVL_LinearActuatorProxSensors.TcGVL
VAR_GLOBAL
	Tri1_Prox_In AT %I* : BOOL;
	Tri1_Prox_Out AT %I* : BOOL;
	Cmp1_Prox_In AT %I* : BOOL;
	Cmp1_Prox_Out AT %I* : BOOL;
	Cmp1_Prox_Fault AT %I* : BOOL;
	Piv1_Prox_In AT %I* : BOOL;
	Piv1_Prox_Out AT %I* : BOOL;
	Tri2_Prox_In AT %I* : BOOL;
	Tri2_Prox_Out AT %I* : BOOL;
	Tri3_Prox_In AT %I* : BOOL;
	Tri3_Prox_Out AT %I* : BOOL;
	Gui1_Prox_In AT %I* : BOOL;
	Gui1_Prox_Out AT %I* : BOOL;
	Gui1_Prox_In_Slow AT %I* : BOOL;
	Gui1_Prox_Out_Slow AT %I* : BOOL;
	Gui2_Prox_In AT %I* : BOOL;
	Gui2_Prox_Out AT %I* : BOOL;
	Gui2_Prox_In_Slow AT %I* : BOOL;
	Gui2_Prox_Out_Slow AT %I* : BOOL;
	Cmp2_Prox_In AT %I* : BOOL;
	Cmp2_Prox_Out AT %I* : BOOL;
	Cmp2_Prox_Fault AT %I* : BOOL;
	Tri4_Prox_In AT %I* : BOOL;
	Tri4_Prox_Out AT %I* : BOOL;
END_VAR

// ---- GVLs/GVL_LinearActuators.TcGVL
VAR_GLOBAL
	
	Tri1_Mot_Struct : ST_LinearActuator := (
		sName := 'Chariot1',
		bProxIn := ADR(Tri1_Prox_In) ,  
		bProxOut := ADR(Tri1_Prox_Out) , 
		bFwdDO := ADR(Tri1_Mot_Fw), 
		bBckwDO := ADR(Tri1_Mot_Bw)
		);
	
	Cmp1_Mot_Struct : ST_LinearActuator := (
		sName := 'Compressor1',
		bProxIn := ADR(Cmp1_Prox_In),  
		bProxOut := ADR(Cmp1_Prox_Out),
		bProx2 := ADR(Cmp1_Prox_Fault),
		bFwdDO := ADR(Cmp1_Mot_Fw), 
		bBckwDO := ADR(Cmp1_Mot_Bw),
		bStopControlDO := ADR(Cmp1_Mot_Stop),
		bFaultDI := ADR(Cmp1_Mot_Fault)
		);
	
	Piv1_Mot_Struct : ST_LinearActuator := (
		sName := 'Sensor1',
		bProxIn := ADR(Piv1_Prox_In),  
		bProxOut := ADR(Piv1_Prox_Out), 
		bFwdDO := ADR(Piv1_Mot_Fw), 
		bBckwDO := ADR(Piv1_Mot_Bw)
		);
	
	Tri2_Mot_Struct : ST_LinearActuator := (
		sName := 'Chariot2',
		bProxIn := ADR(Tri2_Prox_In),  
		bProxOut := ADR(Tri2_Prox_Out), 
		bFwdDO := ADR(Tri2_Mot_Fw), 
		bBckwDO := ADR(Tri2_Mot_Bw)
		);

	Tri3_Mot_Struct : ST_LinearActuator := (
		sName := 'Chariot3',
		bProxIn := ADR(Tri3_Prox_In),  
		bProxOut := ADR(Tri3_Prox_Out), 
		bFwdDO := ADR(Tri3_Mot_Fw), 
		bBckwDO := ADR(Tri3_Mot_Bw)
		);
	
	Gui1_Mot_Struct : ST_LinearActuator := (
		sName := 'HeatExCoupola3',
		bProxIn := ADR(Gui1_Prox_In),  
		bProxOut := ADR(Gui1_Prox_Out),
		bProx2 := ADR(Gui1_Prox_In_Slow),
		bProx3 := ADR(Gui1_Prox_Out_Slow), 
		bFwdDO := ADR(Gui1_Mot_Fw), 
		bBckwDO := ADR(Gui1_Mot_Bw),
		bSpeedControlDO := ADR(Gui1_Mot_Speed2),
		bStopControlDO := ADR(Gui1_Mot_Stop),
		bFaultDI := ADR(Gui1_Mot_Fault)
		);
		
		
	Gui2_Mot_Struct : ST_LinearActuator := (
		sName := 'RegenCoupola3',
		bProxIn := ADR(Gui2_Prox_In),  
		bProxOut := ADR(Gui2_Prox_Out), 
		bProx2 := ADR(Gui2_Prox_In_Slow),
		bProx3 := ADR(Gui2_Prox_Out_Slow), 
		bFwdDO := ADR(Gui2_Mot_Fw), 
		bBckwDO := ADR(Gui2_Mot_Bw),
		bSpeedControlDO := ADR(Gui2_Mot_Speed2),
		bStopControlDO := ADR(Gui2_Mot_Stop),
		bFaultDI := ADR(Gui2_Mot_Fault)
		);
	
	Tri4_Mot_Struct : ST_LinearActuator := (
		sName := 'Chariot4',
		bProxIn := ADR(Tri4_Prox_In),  
		bProxOut := ADR(Tri4_Prox_Out), 
		bFwdDO := ADR(Tri4_Mot_Fw), 
		bBckwDO := ADR(Tri4_Mot_Bw)
		);
	
	Cmp2_Mot_Struct : ST_LinearActuator := (
		sName := 'Compressor3',
		bProxIn := ADR(Cmp2_Prox_In),  
		bProxOut := ADR(Cmp2_Prox_Out),
		bProx2 := ADR(Cmp2_Prox_Fault),
		bFwdDO := ADR(Cmp2_Mot_Fw), 
		bBckwDO := ADR(Cmp2_Mot_Bw),
		bStopControlDO := ADR(Cmp2_Mot_Stop),
		bFaultDI := ADR(Cmp2_Mot_Fault)
		);
	
	Tri1_Mot_FB :  FB_LinearActuator(Actuator := ADR(Tri1_Mot_Struct));
    Cmp1_Mot_FB :  FB_LinearActuator(Actuator := ADR(Cmp1_Mot_Struct));
    Piv1_Mot_FB :  FB_LinearActuator(Actuator := ADR(Piv1_Mot_Struct));
    Tri2_Mot_FB :  FB_LinearActuator(Actuator := ADR(Tri2_Mot_Struct));
    Tri3_Mot_FB :  FB_LinearActuator(Actuator := ADR(Tri3_Mot_Struct));
    Gui1_Mot_FB :  FB_LinearActuator(Actuator := ADR(Gui1_Mot_Struct));
    Gui2_Mot_FB :  FB_LinearActuator(Actuator := ADR(Gui2_Mot_Struct));
	Cmp2_Mot_FB :  FB_LinearActuator(Actuator := ADR(Cmp2_Mot_Struct));
    Tri4_Mot_FB :  FB_LinearActuator(Actuator := ADR(Tri4_Mot_Struct));
	
	Tri1_Mot_Cmd : ST_LinearActuatorCommand;
	Cmp1_Mot_Cmd : ST_LinearActuatorCommand;
	Piv1_Mot_Cmd : ST_LinearActuatorCommand;
	Tri2_Mot_Cmd : ST_LinearACtuatorCommand;
	Tri3_Mot_Cmd : ST_LinearActuatorCommand;
	Gui1_Mot_Cmd : ST_LinearActuatorCommand;
	Gui2_Mot_Cmd : ST_LinearActuatorCommand;
	Tri4_Mot_Cmd : ST_LinearActuatorCommand;
	Cmp2_Mot_Cmd : ST_LinearActuatorCommand; 	
END_VAR

// ---- GVLs/GVL_LinearActuatorRelays.TcGVL
VAR_GLOBAL
	Tri1_Mot_Fw AT %Q* : BOOL; 
	Tri1_Mot_Bw AT %Q* : BOOL; 
	Cmp1_Mot_Fw AT %Q* : BOOL; 
	Cmp1_Mot_Bw AT %Q* : BOOL; 
	Piv1_Mot_Fw AT %Q* : BOOL; 
	Piv1_Mot_Bw AT %Q* : BOOL; 
	Tri2_Mot_Fw AT %Q* : BOOL; 
	Tri2_Mot_Bw AT %Q* : BOOL; 
	Tri3_Mot_Fw AT %Q* : BOOL; 
	Tri3_Mot_Bw AT %Q* : BOOL; 
	Gui1_Mot_Fw AT %Q* : BOOL; 
	Gui1_Mot_Bw AT %Q* : BOOL; 
	Gui2_Mot_Fw AT %Q* : BOOL; 
	Gui2_Mot_Bw AT %Q* : BOOL; 
	Cmp2_Mot_Fw AT %Q* : BOOL; 
	Cmp2_Mot_Bw AT %Q* : BOOL; 
	Tri4_Mot_Fw AT %Q* : BOOL; 
	Tri4_Mot_Bw AT %Q* : BOOL;  
END_VAR

// ---- GVLs/GVL_Process.TcGVL
VAR_GLOBAL
	HeatExchangeRunning: BOOL := FALSE;
	StartHeatExchange: BOOL := FALSE;
	
	AdsorptionRunning: BOOL := FALSE;
	StartAdsorption: BOOL := FALSE;
	
	RegenerationRunning: BOOL := FALSE;
	StartRegeneration: BOOL := FALSE;
END_VAR

// ---- GVLs/GVL_StepperPositions.TcGVL
VAR_GLOBAL
	Rail1_Pos1 : LREAL := 0;
	Rail1_Pos2 : LREAL := 500;
	Rail1_Pos3 : LREAL := 615;
	Rail1_Pos4 : LREAL := 1000;
	Rail1_Pos5 : LREAL := 1205;
	Rail2_Pos1 : LREAL := 0;
	Rail2_Pos2 : LREAL := 955;
	Rail3_Pos1 : LREAL := 45;
	Rail3_Pos2 : LREAL := 145;
	Rail3_Pos3 : LREAL := 600;
	Rail3_Pos4 : LREAL := 645;
	Rail3_Pos5 : LREAL := 1250;
	Rail4_Pos1 : LREAL := 0;
	Rail4_Pos2 : LREAL := 955;	
END_VAR

// ---- POUs/Programs/PRG_Cycle.TcPOU
PROGRAM PRG_Cycle
VAR	
Status : INT := 0;
bHomingDone: BOOL;
fbRTrigStart: INT;
END_VAR

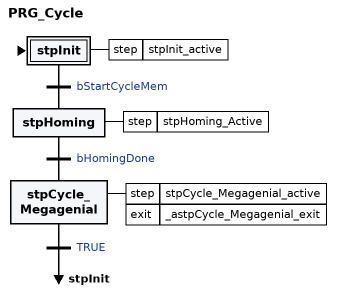
INITIAL_STEP stpInit:
    stpInit_active(N);  // step action
END_STEP
TRANSITION FROM stpInit TO stpHoming
    := bStartCycleMem;
END_TRANSITION
STEP stpHoming:
    stpHoming_Active(N);  // step action
END_STEP
TRANSITION FROM stpHoming TO stpCycle_Megagenial
    := bHomingDone;
END_TRANSITION
STEP stpCycle_Megagenial:
    stpCycle_Megagenial_active(N);  // step action
    _astpCycle_Megagenial_exit(P0);  // exit action
END_STEP
TRANSITION FROM stpCycle_Megagenial TO stpInit
    := TRUE;
END_TRANSITION

ACTION _astpCatch_Rail1_active:
Status := F_IssueActuatorCommand(sDevice := 'R1_Chariot', bArg := TRUE);
END_ACTION

ACTION _astpCatch_Rail2_active:
Status := F_IssueActuatorCommand(sDevice := 'R2_Chariot', bArg := TRUE);
END_ACTION

ACTION _astpCatch_Rail3_active:
Status := F_IssueActuatorCommand(sDevice := 'R3_Chariot', bArg := TRUE);
END_ACTION

ACTION _astpCatch_Rail4_active:
Status := F_IssueActuatorCommand(sDevice := 'R4_Chariot', bArg := TRUE);
END_ACTION

ACTION _astpCycle_Megagenial_exit:
bStartCycleMem := FALSE;
bStopCycleMem := FALSE;
END_ACTION

ACTION _astpDrop_Rail2_active:
Status := F_IssueActuatorCommand(sDevice := 'R2_Chariot', bArg := FALSE);
END_ACTION

ACTION _astpDrop_Rail3_active:
Status := F_IssueActuatorCommand(sDevice := 'R3_Chariot', bArg := FALSE);
END_ACTION

ACTION _astpDrop_Rail4_active:
Status := F_IssueActuatorCommand(sDevice := 'R4_Chariot', bArg := FALSE);
END_ACTION

ACTION _astpHoming_Gui1_active:
Status := F_IssueActuatorCommand(sDevice := 'R3_HeatExCoupola', bArg := FALSE);
END_ACTION

ACTION _astpHoming_Gui2_active:
Status := F_IssueActuatorCommand(sDevice := 'R3_RegenCoupola', bArg := FALSE);
END_ACTION

ACTION _astpHoming_Pous1_active:
Status := F_IssueActuatorCommand(sDevice := 'R1_Compressor', bArg := FALSE);
END_ACTION

ACTION _astpHoming_Pous2_active:
Status := F_IssueActuatorCommand(sDevice := 'R3_Compressor', bArg := FALSE);
END_ACTION

ACTION _astpHoming_Tri1_active:
Status := F_IssueActuatorCommand(sDevice := 'R1_Chariot', bArg := FALSE);
END_ACTION

ACTION _astpHoming_Tri2_active:
Status := F_IssueActuatorCommand(sDevice := 'R2_Chariot', bArg := FALSE);
END_ACTION

ACTION _astpHoming_Tri3_active:
Status := F_IssueActuatorCommand(sDevice := 'R3_Chariot', bArg := FALSE);
END_ACTION

ACTION _astpHoming_Tri4_active:
Status := F_IssueActuatorCommand(sDevice := 'R4_Chariot', bArg := FALSE);
END_ACTION

ACTION _astpMoveBw_Rail1_active:
Status := F_IssueActuatorCommand(sDevice := 'R1_Motor', bArg := FALSE, bHasPosition := TRUE, nPosition:= 100, fVelocity := Mot_LoadedVel);
END_ACTION

ACTION _astpMoveBw_Rail2_active:
Status := F_IssueActuatorCommand(sDevice := 'R2_Motor', bArg := FALSE, bHasPosition := TRUE, nPosition:= 100, fVelocity := Mot_LoadedVel);
END_ACTION

ACTION _astpMoveBw_Rail3_active:
Status := F_IssueActuatorCommand(sDevice := 'R3_Motor', bArg := FALSE, bHasPosition := TRUE, nPosition:= 100, fVelocity := Mot_LoadedVel);
END_ACTION

ACTION _astpMoveBw_Rail4_active:
Status := F_IssueActuatorCommand(sDevice := 'R4_Motor', bArg := FALSE, bHasPosition := TRUE, nPosition:= 100, fVelocity := Mot_LoadedVel);
END_ACTION

ACTION _astpMoveFw_Rail1_active:
Status := F_IssueActuatorCommand(sDevice := 'R1_Motor', bArg := FALSE, bHasPosition := TRUE, nPosition:= 1295, fVelocity := Mot_UnloadedVel);
END_ACTION

ACTION _astpMoveFw_Rail2_active:
Status := F_IssueActuatorCommand(sDevice := 'R2_Motor', bArg := FALSE, bHasPosition := TRUE, nPosition:= 980, fVelocity := Mot_UnloadedVel);
END_ACTION

ACTION _astpMoveFw_Rail3_active:
Status := F_IssueActuatorCommand(sDevice := 'R3_Motor', bArg := FALSE, bHasPosition := TRUE, nPosition:= 1295, fVelocity := Mot_UnloadedVel);
END_ACTION

ACTION _astpMoveFw_Rail4_active:
Status := F_IssueActuatorCommand(sDevice := 'R4_Motor', bArg := FALSE, bHasPosition := TRUE, nPosition:= 1295, fVelocity := Mot_UnloadedVel);
END_ACTION

ACTION stpCycle_Megagenial_active:
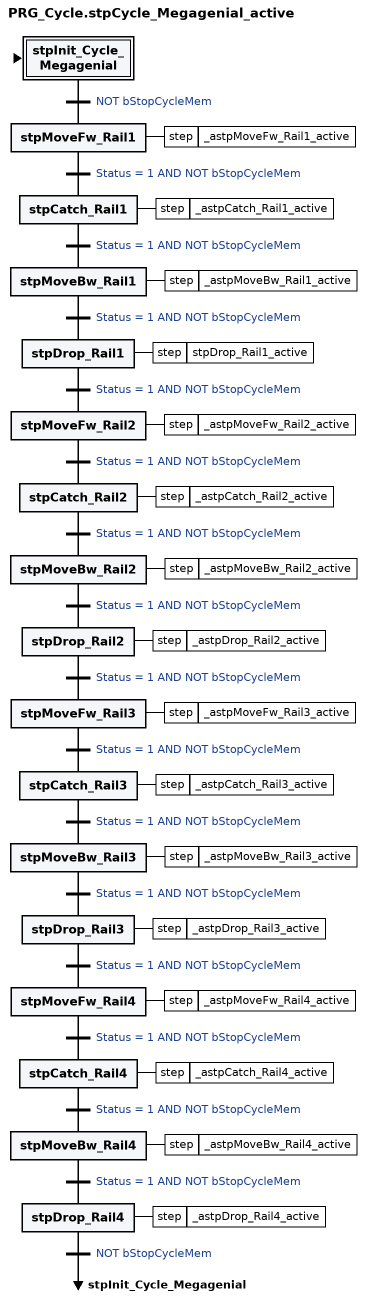
INITIAL_STEP stpInit_Cycle_Megagenial:
END_STEP
TRANSITION FROM stpInit_Cycle_Megagenial TO stpMoveFw_Rail1
    := NOT bStopCycleMem;
END_TRANSITION
STEP stpMoveFw_Rail1:
    _astpMoveFw_Rail1_active(N);  // step action
END_STEP
TRANSITION FROM stpMoveFw_Rail1 TO stpCatch_Rail1
    := Status = 1 AND NOT bStopCycleMem;
END_TRANSITION
STEP stpCatch_Rail1:
    _astpCatch_Rail1_active(N);  // step action
END_STEP
TRANSITION FROM stpCatch_Rail1 TO stpMoveBw_Rail1
    := Status = 1 AND NOT bStopCycleMem;
END_TRANSITION
STEP stpMoveBw_Rail1:
    _astpMoveBw_Rail1_active(N);  // step action
END_STEP
TRANSITION FROM stpMoveBw_Rail1 TO stpDrop_Rail1
    := Status = 1 AND NOT bStopCycleMem;
END_TRANSITION
STEP stpDrop_Rail1:
    stpDrop_Rail1_active(N);  // step action
END_STEP
TRANSITION FROM stpDrop_Rail1 TO stpMoveFw_Rail2
    := Status = 1 AND NOT bStopCycleMem;
END_TRANSITION
STEP stpMoveFw_Rail2:
    _astpMoveFw_Rail2_active(N);  // step action
END_STEP
TRANSITION FROM stpMoveFw_Rail2 TO stpCatch_Rail2
    := Status = 1 AND NOT bStopCycleMem;
END_TRANSITION
STEP stpCatch_Rail2:
    _astpCatch_Rail2_active(N);  // step action
END_STEP
TRANSITION FROM stpCatch_Rail2 TO stpMoveBw_Rail2
    := Status = 1 AND NOT bStopCycleMem;
END_TRANSITION
STEP stpMoveBw_Rail2:
    _astpMoveBw_Rail2_active(N);  // step action
END_STEP
TRANSITION FROM stpMoveBw_Rail2 TO stpDrop_Rail2
    := Status = 1 AND NOT bStopCycleMem;
END_TRANSITION
STEP stpDrop_Rail2:
    _astpDrop_Rail2_active(N);  // step action
END_STEP
TRANSITION FROM stpDrop_Rail2 TO stpMoveFw_Rail3
    := Status = 1 AND NOT bStopCycleMem;
END_TRANSITION
STEP stpMoveFw_Rail3:
    _astpMoveFw_Rail3_active(N);  // step action
END_STEP
TRANSITION FROM stpMoveFw_Rail3 TO stpCatch_Rail3
    := Status = 1 AND NOT bStopCycleMem;
END_TRANSITION
STEP stpCatch_Rail3:
    _astpCatch_Rail3_active(N);  // step action
END_STEP
TRANSITION FROM stpCatch_Rail3 TO stpMoveBw_Rail3
    := Status = 1 AND NOT bStopCycleMem;
END_TRANSITION
STEP stpMoveBw_Rail3:
    _astpMoveBw_Rail3_active(N);  // step action
END_STEP
TRANSITION FROM stpMoveBw_Rail3 TO stpDrop_Rail3
    := Status = 1 AND NOT bStopCycleMem;
END_TRANSITION
STEP stpDrop_Rail3:
    _astpDrop_Rail3_active(N);  // step action
END_STEP
TRANSITION FROM stpDrop_Rail3 TO stpMoveFw_Rail4
    := Status = 1 AND NOT bStopCycleMem;
END_TRANSITION
STEP stpMoveFw_Rail4:
    _astpMoveFw_Rail4_active(N);  // step action
END_STEP
TRANSITION FROM stpMoveFw_Rail4 TO stpCatch_Rail4
    := Status = 1 AND NOT bStopCycleMem;
END_TRANSITION
STEP stpCatch_Rail4:
    _astpCatch_Rail4_active(N);  // step action
END_STEP
TRANSITION FROM stpCatch_Rail4 TO stpMoveBw_Rail4
    := Status = 1 AND NOT bStopCycleMem;
END_TRANSITION
STEP stpMoveBw_Rail4:
    _astpMoveBw_Rail4_active(N);  // step action
END_STEP
TRANSITION FROM stpMoveBw_Rail4 TO stpDrop_Rail4
    := Status = 1 AND NOT bStopCycleMem;
END_TRANSITION
STEP stpDrop_Rail4:
    _astpDrop_Rail4_active(N);  // step action
END_STEP
TRANSITION FROM stpDrop_Rail4 TO stpInit_Cycle_Megagenial
    := NOT bStopCycleMem;
END_TRANSITION
END_ACTION

ACTION stpDrop_Rail1_active:
Status := F_IssueActuatorCommand(sDevice := 'R1_Chariot', bArg := FALSE);
END_ACTION

ACTION stpHoming_Active:
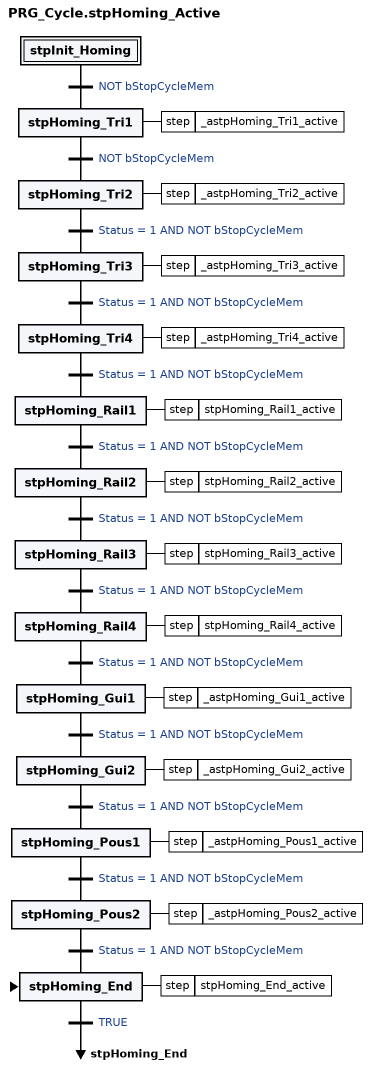
INITIAL_STEP stpInit_Homing:
END_STEP
TRANSITION FROM stpInit_Homing TO stpHoming_Tri1
    := NOT bStopCycleMem;
END_TRANSITION
STEP stpHoming_Tri1:
    _astpHoming_Tri1_active(N);  // step action
END_STEP
TRANSITION FROM stpHoming_Tri1 TO stpHoming_Tri2
    := NOT bStopCycleMem;
END_TRANSITION
STEP stpHoming_Tri2:
    _astpHoming_Tri2_active(N);  // step action
END_STEP
TRANSITION FROM stpHoming_Tri2 TO stpHoming_Tri3
    := Status = 1 AND NOT bStopCycleMem;
END_TRANSITION
STEP stpHoming_Tri3:
    _astpHoming_Tri3_active(N);  // step action
END_STEP
TRANSITION FROM stpHoming_Tri3 TO stpHoming_Tri4
    := Status = 1 AND NOT bStopCycleMem;
END_TRANSITION
STEP stpHoming_Tri4:
    _astpHoming_Tri4_active(N);  // step action
END_STEP
TRANSITION FROM stpHoming_Tri4 TO stpHoming_Rail1
    := Status = 1 AND NOT bStopCycleMem;
END_TRANSITION
STEP stpHoming_Rail1:
    stpHoming_Rail1_active(N);  // step action
END_STEP
TRANSITION FROM stpHoming_Rail1 TO stpHoming_Rail2
    := Status = 1 AND NOT bStopCycleMem;
END_TRANSITION
STEP stpHoming_Rail2:
    stpHoming_Rail2_active(N);  // step action
END_STEP
TRANSITION FROM stpHoming_Rail2 TO stpHoming_Rail3
    := Status = 1 AND NOT bStopCycleMem;
END_TRANSITION
STEP stpHoming_Rail3:
    stpHoming_Rail3_active(N);  // step action
END_STEP
TRANSITION FROM stpHoming_Rail3 TO stpHoming_Rail4
    := Status = 1 AND NOT bStopCycleMem;
END_TRANSITION
STEP stpHoming_Rail4:
    stpHoming_Rail4_active(N);  // step action
END_STEP
TRANSITION FROM stpHoming_Rail4 TO stpHoming_Gui1
    := Status = 1 AND NOT bStopCycleMem;
END_TRANSITION
STEP stpHoming_Gui1:
    _astpHoming_Gui1_active(N);  // step action
END_STEP
TRANSITION FROM stpHoming_Gui1 TO stpHoming_Gui2
    := Status = 1 AND NOT bStopCycleMem;
END_TRANSITION
STEP stpHoming_Gui2:
    _astpHoming_Gui2_active(N);  // step action
END_STEP
TRANSITION FROM stpHoming_Gui2 TO stpHoming_Pous1
    := Status = 1 AND NOT bStopCycleMem;
END_TRANSITION
STEP stpHoming_Pous1:
    _astpHoming_Pous1_active(N);  // step action
END_STEP
TRANSITION FROM stpHoming_Pous1 TO stpHoming_Pous2
    := Status = 1 AND NOT bStopCycleMem;
END_TRANSITION
STEP stpHoming_Pous2:
    _astpHoming_Pous2_active(N);  // step action
END_STEP
TRANSITION FROM stpHoming_Pous2 TO stpHoming_End
    := Status = 1 AND NOT bStopCycleMem;
END_TRANSITION
STEP stpHoming_End:
    stpHoming_End_active(N);  // step action
END_STEP
TRANSITION FROM stpHoming_End TO stpHoming_End
    := TRUE;
END_TRANSITION
END_ACTION

ACTION stpHoming_End_active:
bHomingDone := TRUE;
END_ACTION

ACTION stpHoming_Rail1_active:
Status := F_IssueActuatorCommand(sDevice := 'R1_Motor', bArg := TRUE);
END_ACTION

ACTION stpHoming_Rail2_active:
Status := F_IssueActuatorCommand(sDevice := 'R2_Motor', bArg := TRUE);
END_ACTION

ACTION stpHoming_Rail3_active:
Status := F_IssueActuatorCommand(sDevice := 'R3_Motor', bArg := TRUE);
END_ACTION

ACTION stpHoming_Rail4_active:
Status := F_IssueActuatorCommand(sDevice := 'R4_Motor', bArg := TRUE);
END_ACTION

ACTION stpInit_active:
RTrigStart(CLK := StartCycle OR StartCycle_HMI);
RTrigStop (CLK := StopCycle OR StopCycle_HMI);

(* If START is pressed -> remember START, forget STOP *)
IF RTrigStart.Q THEN
    bStartCycleMem := TRUE;
    bStopCycleMem  := FALSE;
END_IF

(* If STOP is pressed -> remember STOP, forget START *)
IF RTrigStop.Q THEN
    bStopCycleMem  := TRUE;
    bStartCycleMem := FALSE;
END_IF
END_ACTION

END_PROGRAM

// ---- POUs/Helper/F_IssueActuatorCommand.TcPOU
FUNCTION F_IssueActuatorCommand : INT
VAR_INPUT
    sDevice       : STRING(50);   // e.g. 'Chariot1', 'Motor3', ...
    bArg          : BOOL;         // see spec: direction or homing flag
    bHasPosition  : BOOL := FALSE;
    nPosition     : LREAL := 0;    // used when Motor & !bArg & position present
	fVelocity    : LREAL := 100.0;
END_VAR
VAR
    nlen       : INT;
    n         : INT;
    sPrefix   : STRING(50);
    i         : INT;
    sTmp      : STRING(64);
    sIndexStr : STRING(1);
END_VAR

(* ---- basic checks ---- *)
nLen := LEN(sDevice);
IF nLen < 2 THEN
    F_IssueActuatorCommand := -1;
    RETURN;
END_IF;

// last digit "1".."4"
sIndexStr := MID(sDevice, 1, nLen);      // 1 char at position nLen
n := STRING_TO_INT(sIndexStr);

// prefix = everything except last char
sPrefix := LEFT(sDevice, nLen - 1);

(* ---- build "R<n>_" into sTmp ---- *)
sTmp := CONCAT('R', INT_TO_STRING(n));
sTmp := CONCAT(sTmp, '_');

(* ===================== *)
(* Non-motor devices     *)
(* ===================== *)
IF (sPrefix = 'Chariot') OR (sPrefix = 'Compressor') OR (sPrefix = 'Sensor') OR
   (sPrefix = 'HeatExCoupola') OR (sPrefix = 'RegenCoupola') THEN

    sRequestedActuator := CONCAT(sTmp, sPrefix);   // "R<n>_Prefix"

    IF sPrefix = 'Chariot' THEN
        CASE n OF
            1: Tri1_Mot_Cmd.bCommand := bArg;
            2: Tri2_Mot_Cmd.bCommand := bArg;
            3: Tri3_Mot_Cmd.bCommand := bArg;
            4: Tri4_Mot_Cmd.bCommand := bArg;
        END_CASE

    ELSIF sPrefix = 'Compressor' THEN
        CASE n OF
            1: Cmp1_Mot_Cmd.bCommand := bArg;
            3: Cmp2_Mot_Cmd.bCommand := bArg;
            (* n=2,4 handled elsewhere if needed *)
        END_CASE

    ELSIF sPrefix = 'Sensor' THEN
        CASE n OF
            1: Piv1_Mot_Cmd.bCommand := bArg;
        END_CASE

    ELSIF sPrefix = 'HeatExCoupola' THEN
        CASE n OF
            3: Gui1_Mot_Cmd.bCommand := bArg;
        END_CASE

    ELSIF sPrefix = 'RegenCoupola' THEN
        CASE n OF
            3: Gui2_Mot_Cmd.bCommand := bArg;
        END_CASE
    END_IF;

    // <<< return handling for non-motor >>>
    // function returns the global Result:
    //   -1 = failure, 0 = in progress, 1 = success
    F_IssueActuatorCommand := Result;
    RETURN;
END_IF

(* ===================== *)
(* Motor devices         *)
(* ===================== *)
IF sPrefix = 'Motor' THEN
    
    IF bArg THEN
        (* Homing *)
        sRequestedActuator := CONCAT(sTmp, 'Home');   // "R<n>_Home"
        CASE n OF
            1: Rail1_Mot_Cmd.bHoming := TRUE;
            2: Rail2_Mot_Cmd.bHoming := TRUE;
            3: Rail3_Mot_Cmd.bHoming := TRUE;
            4: Rail4_Mot_Cmd.bHoming := TRUE;
        END_CASE
    ELSE
        (* Normal move *)
        sRequestedActuator := CONCAT(sTmp, 'Motor');  // "R<n>_Motor"
        
        IF bHasPosition THEN
            CASE n OF
                1: 
                    Rail1_Mot_Cmd.nCommand := nPosition;
                    (* Velocity Logic *)
                    IF fVelocity > 0.0 THEN
                        Rail1_Mot_Cmd.fVelocity := fVelocity;
                    ELSE
                        Rail1_Mot_Cmd.fVelocity := Mot_LoadedVel;
                    END_IF;

                2: 
                    Rail2_Mot_Cmd.nCommand := nPosition;
                    IF fVelocity > 0.0 THEN
                        Rail2_Mot_Cmd.fVelocity := fVelocity;
                    ELSE
                        Rail2_Mot_Cmd.fVelocity := Mot_LoadedVel;
                    END_IF;

                3: 
                    Rail3_Mot_Cmd.nCommand := nPosition;
                    IF fVelocity > 0.0 THEN
                        Rail3_Mot_Cmd.fVelocity := fVelocity;
                    ELSE
                        Rail3_Mot_Cmd.fVelocity := Mot_LoadedVel;
                    END_IF;

                4: 
                    Rail4_Mot_Cmd.nCommand := nPosition;
                    IF fVelocity > 0.0 THEN
                        Rail4_Mot_Cmd.fVelocity := fVelocity;
                    ELSE
                        Rail4_Mot_Cmd.fVelocity := Mot_LoadedVel;
                    END_IF;
            END_CASE
        END_IF
    END_IF;

    // <<< return handling for motors >>>
    F_IssueActuatorCommand := Result; // Assuming 'Result' is defined globally or earlier
    RETURN;
END_IF

(* Unknown prefix *)
F_IssueActuatorCommand := -3;

END_FUNCTION

// ---- POUs/Programs/PRG_AlarmHandler.TcPOU
PROGRAM PRG_AlarmHandler
VAR
    fbAlarmStatusManager : FB_AlarmStatusManager;
	bInitComplete : BOOL := FALSE;

	nIndex : SINT;
	fbFlashTimerStart : TON;
	bFlashStateStart  : BOOL;
	
	fbFlashTimerStop : TON;
	bFlashStateStop  : BOOL;
	
	(* MAINTENANCE MODE TOGGLE *)
    bMaintenanceMode : BOOL := FALSE;
END_VAR

(* Rail number Init *)
IF NOT bInitComplete THEN
    Rail1_Mot_FB.nRail := 1;
    Rail2_Mot_FB.nRail := 2; 
    Rail3_Mot_FB.nRail := 3;
    Rail4_Mot_FB.nRail := 4;
	
    bInitComplete := TRUE;
END_IF

(* Read physical door and HMI inputs *)
RTrigStart(CLK := StartCycle OR StartCycle_HMI);
RTrigStop (CLK := StopCycle OR StopCycle_HMI);
RTrigReset(CLK := bResetSafety);
	
IF RTrigStart.Q THEN
    bStartCycleMem := TRUE;   
    StartCycle_HMI := FALSE; 
END_IF

IF RTrigStop.Q THEN
    bStopCycleMem  := TRUE;
    StopCycle_HMI := FALSE;
END_IF

IF RTrigReset.Q THEN
    bResetSafetyMem := TRUE;
END_IF

(* Start LED flash *)
IF bSafetyOk AND NOT bStartCycleMem THEN
	fbFlashTimerStart (IN := NOT fbFlashTimerStart .Q, PT := T#250MS);

	IF fbFlashTimerStart .Q THEN
		bFlashStateStart  := NOT bFlashStateStart ;
	END_IF

	bStartLED := bFlashStateStart ;
ELSIF bStartCycleMem AND bSafetyOk THEN
	bStartLED := TRUE;
ELSE
	bStartLED := FALSE;
END_IF

(* Stop LED flash *)
IF bStopCycleMem AND NOT bCycleDone THEN
	fbFlashTimerStop(IN := NOT fbFlashTimerStop .Q, PT := T#250MS);

	IF fbFlashTimerStop .Q THEN
		bFlashStateStop  := NOT bFlashStateStop ;
	END_IF

	bStopLED := bFlashStateStop ;
ELSE
	bStopLED := FALSE;
END_IF

(* If Safety is triggered but command doesnt return -1 in cycle, force it *)
IF NOT bSafetyOk AND bStartCycleMem THEN
	bSFCResetCommand^ := TRUE;
	bStopCycleMem := FALSE;
	bStartCycleMem := FALSE;
	bHomingDone := FALSE;
	bCycleDone := FALSE;
	Result := 0;
END_IF

fbAlarmStatusManager(bMaintenanceMode := bMaintenanceMode);
gSystemAlarmStatus := fbAlarmStatusManager.stSystemStatus;

END_PROGRAM

// ---- POUs/FunctionBlocks/FB_AlarmStatusManager.TcPOU
FUNCTION_BLOCK FB_AlarmStatusManager
VAR_INPUT
    bMaintenanceMode : BOOL;  
END_VAR

VAR_OUTPUT
    stSystemStatus : ST_SystemAlarmStatus;  
END_VAR

VAR
    i : INT;
    bFirstRun : BOOL := TRUE;
    nZone : SINT;
    bIsGlobalAlarm : BOOL;
	
	nMainState    : INT := 0;   (* Controls the flow of the repetitions *)
	nRepetition   : INT := 0;   (* Counts how many times we have finished the sequence *)
	nStep : INT := 1;
    aAllAlarms : ARRAY[1..100] OF ST_AlarmEntry;
    nAlarmCount : INT := 0;
	fbFlashTimer : TON;
	bFlashState  : BOOL;
END_VAR

stSystemStatus.bMaintenanceMode := bMaintenanceMode;

// Initialize alarm list 
IF bFirstRun THEN
    InitializeAlarmList();
    bFirstRun := FALSE;
END_IF

// Reset all zones to OK
bCriticalAlarm := FALSE;

FOR i := 1 TO 5 DO
    stSystemStatus.aZoneStatus[i].bOkToRun := TRUE;
    stSystemStatus.aZoneStatus[i].nHighestSeverity := 0;
END_FOR

//Check Safety Relay status
SafetyRelay.bCondition := NOT SafetyRelayStatus;

IF SafetyRelay.bCondition THEN
	(* Timer counts to 250ms, then resets itself *)
	fbFlashTimer(IN := NOT fbFlashTimer.Q, PT := T#250MS);

	(* Every time the timer finishes (Q=TRUE), toggle the state *)
	IF fbFlashTimer.Q THEN
		bFlashState := NOT bFlashState;
	END_IF

	(* Map to your physical output *)
	bResetLED := bFlashState;
ELSE
	bResetLED := FALSE;
END_IF

HandlePhysicalResetReq();

// Process all alarms 
FOR i := 1 TO nAlarmCount DO
    IF aAllAlarms[i].pAlarm <> 0 THEN
		nZone := ParseAlarmZone(aAllAlarms[i].sName);
		ProcessAlarm(aAllAlarms[i].pAlarm, nZone);	
    END_IF
	
END_FOR

METHOD AddAlarm : BOOL
VAR_INPUT
    pAlarm : POINTER TO ST_Alarm;
    sAlarmName : STRING(50);
END_VAR
nAlarmCount := nAlarmCount + 1;
aAllAlarms[nAlarmCount].pAlarm := pAlarm;
aAllAlarms[nAlarmCount].sName := sAlarmName;

AddAlarm := TRUE;
END_METHOD

METHOD HandlePhysicalResetReq : BOOL
VAR
	nOutput : INT;
	fbLoopTimer   : TON;        (* The 1s timer between loops *)
END_VAR
IF bSafetyOk THEN
	bResetSafetyMem := FALSE;
END_IF

IF bResetSafetyMem AND NOT bCriticalAlarm AND NOT bSafetyOk THEN
    CASE nMainState OF
        0: (* INITIALIZATION *)
            nRepetition := 0;
            nStep := 1;          (* Ensure motors start at 1 *)
            nMainState := 10;    (* Start the sequence *)

        10: (* EXECUTE THE 4 STEPS (Your Original Logic) *)
            
            CASE nStep OF
                1: sRequestedActuator := 'R1_Motor_Reset';
                2: sRequestedActuator := 'R2_Motor_Reset';
                3: sRequestedActuator := 'R3_Motor_Reset';
                4: sRequestedActuator := 'R4_Motor_Reset';
            END_CASE
            
            nOutput := Result;
            
            CASE nOutput OF
                1:  nStep := nStep + 1; (* Success, next motor *)
                0:  RETURN;             (* Still working, wait *)
                -1: nStep := nStep + 1; (* Error, skip to next *)
            END_CASE
            
            (* WHEN ALL 4 MOTORS ARE DONE *)
            IF nStep > 4 THEN
                nMainState := 20; (* Don't finish yet! Go to the waiting state. *)
            END_IF

        20: (* WAIT 1 SECOND *)
            fbLoopTimer(IN := TRUE, PT := T#1S);
            
            IF fbLoopTimer.Q THEN
                (* 1 Second has passed *)
                fbLoopTimer(IN := FALSE);       (* Reset timer *)
                nRepetition := nRepetition + 1; (* Count this run *)
                
                (* CHECK IF WE ARE DONE *)
                IF nRepetition < 4 THEN
                    nStep := 1;       (* Reset motors to start *)
                    nMainState := 10; (* Go back and run them again *)
                ELSE
                    nMainState := 30; (* We have done 4 runs, finish up *)
                END_IF
            END_IF

        30: (* FINISH *)
            bResetSafetyMem := FALSE; (* Turn off the master trigger *)
            nMainState := 0;          (* Reset state for next time safety is pressed *)
            
    END_CASE

ELSE
    (* Safety precaution: Reset everything if the trigger condition is lost *)
    nMainState := 0;
    fbLoopTimer(IN := FALSE);
END_IF
END_METHOD

METHOD InitializeAlarmList : BOOL
nAlarmCount := 0;

(* RAIL 1 *)
AddAlarm(ADR(GVL_Alarms.R1_Sensor_UnknownPosition), 'R1_Sensor_UnknownPosition');
AddAlarm(ADR(GVL_Alarms.R1_Sensor_MotionTimedOut), 'R1_Sensor_MotionTimedOut');
AddAlarm(ADR(GVL_Alarms.R1_Compressor_UnknownPosition), 'R1_Compressor_UnknownPosition');
AddAlarm(ADR(GVL_Alarms.R1_Compressor_MotionTimedOut), 'R1_Compressor_MotionTimedOut');
AddAlarm(ADR(GVL_Alarms.R1_Chariot_MotionTimedOut), 'R1_Chariot_MotionTimedOut');
AddAlarm(ADR(GVL_Alarms.R1_Chariot_UnknownPosition), 'R1_Chariot_UnknownPosition');
AddAlarm(ADR(GVL_Alarms.R1_Stepper_Motion_Failed), 'R1_Stepper_Motion_Failed');
AddAlarm(ADR(GVL_Alarms.R1_Stepper_Homing_Failed), 'R1_Stepper_Homing_Failed');
AddAlarm(ADR(GVL_Alarms.R1_Stepper_Motion_Interrupted), 'R1_Stepper_Motion_Interrupted');
AddAlarm(ADR(GVL_Alarms.R1_Stepper_PowerUp_Failed), 'R1_Stepper_PowerUp_Failed');
AddAlarm(ADR(GVL_Alarms.R1_Stepper_Reset_Failed), 'R1_Stepper_Reset_Failed');
AddAlarm(ADR(GVL_Alarms.R1_Stepper_Stop_Failed), 'R1_Stepper_Stop_Failed');
AddAlarm(ADR(GVL_Alarms.R1_Stepper_UnableToReadPosition), 'R1_Stepper_UnableToReadPosition');

(* RAIL 2 *)
AddAlarm(ADR(GVL_Alarms.R2_Stepper_PowerUp_Failed), 'R2_Stepper_PowerUp_Failed');
AddAlarm(ADR(GVL_Alarms.R2_Stepper_Homing_Failed), 'R2_Stepper_Homing_Failed');
AddAlarm(ADR(GVL_Alarms.R2_Stepper_Motion_Failed), 'R2_Stepper_Motion_Failed');
AddAlarm(ADR(GVL_Alarms.R2_Stepper_Motion_Interrupted), 'R2_Stepper_Motion_Interrupted');
AddAlarm(ADR(GVL_Alarms.R2_Stepper_Reset_Failed), 'R2_Stepper_Reset_Failed');
AddAlarm(ADR(GVL_Alarms.R2_Chariot_UnknownPosition), 'R2_Chariot_UnknownPosition');
AddAlarm(ADR(GVL_Alarms.R2_Chariot_MotionTimedOut), 'R2_Chariot_MotionTimedOut');
AddAlarm(ADR(GVL_Alarms.R2_Stepper_Stop_Failed), 'R2_Stepper_Stop_Failed');
AddAlarm(ADR(GVL_Alarms.R2_Stepper_UnableToReadPosition), 'R2_Stepper_UnableToReadPosition');

(* RAIL 3 *)
AddAlarm(ADR(GVL_Alarms.R3_Compressor_UnknownPosition), 'R3_Compressor_UnknownPosition');
AddAlarm(ADR(GVL_Alarms.R3_HeatExCoupola_DriveFaulted), 'R3_HeatExCoupola_DriveFaulted');
AddAlarm(ADR(GVL_Alarms.R3_RegenCoupola_DriveFaulted), 'R3_RegenCoupola_DriveFaulted');
AddAlarm(ADR(GVL_Alarms.R3_Compressor_MotionTimedOut), 'R3_Compressor_MotionTimedOut');
AddAlarm(ADR(GVL_Alarms.R3_HeatExCoupola_UnknownState), 'R3_HeatExCoupola_UnknownPosition');
AddAlarm(ADR(GVL_Alarms.R3_HeatExCoupola_MotionTimedOut), 'R3_HeatExCoupola_MotionTimedOut');
AddAlarm(ADR(GVL_Alarms.R3_RegenCoupola_UnknownPosition), 'R3_RegenCoupola_UnknownPosition');
AddAlarm(ADR(GVL_Alarms.R3_RegenCoupola_MotionTimedOut), 'R3_RegenCoupola_MotionTimedOut');
AddAlarm(ADR(GVL_Alarms.R3_Chariot_UnknownPosition), 'R3_Chariot_UnknownPosition');
AddAlarm(ADR(GVL_Alarms.R3_Chariot_MotionTimedOut), 'R3_Chariot_MotionTimedOut');
AddAlarm(ADR(GVL_Alarms.R3_Stepper_PowerUp_Failed), 'R3_Stepper_PowerUp_Failed');
AddAlarm(ADR(GVL_Alarms.R3_Stepper_Homing_Failed), 'R3_Stepper_Homing_Failed');
AddAlarm(ADR(GVL_Alarms.R3_Stepper_Motion_Failed), 'R3_Stepper_Motion_Failed');
AddAlarm(ADR(GVL_Alarms.R3_Stepper_Motion_Interrupted), 'R3_Stepper_Motion_Interrupted');
AddAlarm(ADR(GVL_Alarms.R3_Stepper_Reset_Failed), 'R3_Stepper_Reset_Failed');
AddAlarm(ADR(GVL_Alarms.R3_Stepper_Stop_Failed), 'R3_Stepper_Stop_Failed');
AddAlarm(ADR(GVL_Alarms.R3_Stepper_UnableToReadPosition), 'R3_Stepper_UnableToReadPosition');

(* RAIL 4 *)
AddAlarm(ADR(GVL_Alarms.R4_Stepper_PowerUp_Failed), 'R4_Stepper_PowerUp_Failed');
AddAlarm(ADR(GVL_Alarms.R4_Stepper_Homing_Failed), 'R4_Stepper_Homing_Failed');
AddAlarm(ADR(GVL_Alarms.R4_Stepper_Motion_Failed), 'R4_Stepper_Motion_Failed');
AddAlarm(ADR(GVL_Alarms.R4_Stepper_Motion_Interrupted), 'R4_Stepper_Motion_Interrupted');
AddAlarm(ADR(GVL_Alarms.R4_Stepper_Reset_Failed), 'R4_Stepper_Reset_Failed');
AddAlarm(ADR(GVL_Alarms.R4_Chariot_UnknownPosition), 'R4_Chariot_UnknownPosition');
AddAlarm(ADR(GVL_Alarms.R4_Chariot_MotionTimedOut), 'R4_Chariot_MotionTimedOut');
AddAlarm(ADR(GVL_Alarms.R4_Stepper_Stop_Failed), 'R4_Stepper_Stop_Failed');
AddAlarm(ADR(GVL_Alarms.R4_Stepper_UnableToReadPosition), 'R4_Stepper_UnableToReadPosition');

(* GLOBAL SECURITY *)
AddAlarm(ADR(GVL_Alarms.SafetyRelay), 'SafetyRelay');
InitializeAlarmList := TRUE;
END_METHOD

METHOD ParseAlarmZone : SINT
VAR_INPUT
    sAlarmName : STRING(50);
END_VAR
VAR
    sZoneChar : STRING(1);
    nZoneNum : SINT;
    sAfterR : STRING;
END_VAR
ParseAlarmZone := 0;

// Check if alarm is global or belongs to a zone
IF LEN(sAlarmName) >= 3 AND LEFT(sAlarmName, 1) = 'R' THEN

    sAfterR := RIGHT(sAlarmName, LEN(sAlarmName) - 1);
    
    sZoneChar := LEFT(sAfterR, 1);
    nZoneNum := STRING_TO_SINT(sZoneChar);
    
    IF nZoneNum >= 1 AND nZoneNum <= 4 AND LEFT(RIGHT(sAfterR, LEN(sAfterR) - 1), 1) = '_' THEN
        ParseAlarmZone := nZoneNum;
    END_IF
	
ELSE
    ParseAlarmZone := 5;  
END_IF
END_METHOD

METHOD ProcessAlarm : BOOL
VAR_INPUT
    pAlarm : POINTER TO ST_Alarm;
    nZone : SINT;
END_VAR
VAR
    nSeverity : UINT;
    bAlarmActive : BOOL;
END_VAR
// Check validity
IF pAlarm = 0 OR nZone < 1 OR nZone > 5 THEN
    ProcessAlarm := FALSE;
    RETURN;
END_IF

nSeverity := pAlarm^.nSeverity;
bAlarmActive := pAlarm^.bCondition;  

IF bAlarmActive THEN
    IF nSeverity > stSystemStatus.aZoneStatus[nZone].nHighestSeverity THEN
        stSystemStatus.aZoneStatus[nZone].nHighestSeverity := nSeverity;
    END_IF

    CASE nSeverity OF
        1, 2: // Info, Warning - No blocking 
            
        3, 4: // Error - Block unless maintenance mode
            IF NOT bMaintenanceMode THEN
                stSystemStatus.aZoneStatus[nZone].bOkToRun := FALSE;
            END_IF
            
        5: // Critical 
            stSystemStatus.aZoneStatus[nZone].bOkToRun := FALSE;
			bCriticalAlarm := TRUE;
    END_CASE
END_IF

ProcessAlarm := TRUE;
END_METHOD

END_FUNCTION_BLOCK

// ---- POUs/Programs/PRG_CommandHandler.TcPOU
PROGRAM PRG_CommandHandler
VAR
    // COMMAND & STATE FLAGS
	bCanProcessCommand    : BOOL;
    bisValidCmd           : BOOL;
    bCancelCmd            : BOOL;
    bHome                 : BOOL;
    bisLinearActuator     : BOOL;
    bisLinearTableHomeCmd : BOOL;
	bisLinearTableSetHomeCmd : BOOL;
    bisLinearTableMoveCmd : BOOL;
    bisResetCmd           : BOOL;

    bOperationInProgress  : BOOL := FALSE;
    bCancelInProgress     : BOOL := FALSE;
    CancelMove            : BOOL := FALSE;
    bSafetyOk             : BOOL := FALSE;
    bAwaitingHMIClose     : BOOL := FALSE;

    // REFERENCES TO FUNCTION BLOCKS / STRUCTURES
    LinearActuator    : POINTER TO FB_LinearActuator;
    LinearTable       : POINTER TO FB_StepperMotor;
    LinearActuatorCmd : POINTER TO ST_LinearActuatorCommand;
    LinearTableCmd    : POINTER TO ST_StepperMotorCommand;

    // INPUTS / PARAMETERS
    nX                 : SINT;
    sY                 : STRING;
    sZ                 : STRING;

    // OUTPUTS / RESULTS
    CurrentPosition : LREAL;

    // LOOP / TEMP VARIABLES
    i : INT;

    // TIMERS
    tmrCancelTimeout   : TON;
    tCancelTimeout     : TIME := T#5S;

    tmrHMICloseSignal  : TON;
    tHMICloseHoldTime  : TIME := T#2000MS;
END_VAR

(* 1. SAFETY CHECK *)
bSafetyOk := EvaluateSystemSafety();

(* 2. WAIT FOR HMI TO EXIT COMMAND PROMPT IF NEEDED*)
IF bAwaitingHMIClose THEN
    tmrHMICloseSignal(IN := TRUE, PT := tHMICloseHoldTime);
    
    IF tmrHMICloseSignal.Q THEN     
        sRequestedActuator := 'none';
        bAwaitingHMIClose := FALSE;
        tmrHMICloseSignal(IN := FALSE);
    END_IF
    
    RETURN;
END_IF

(* 3. COMMAND CANCEL CHECK *)
IF CancelMove AND bOperationInProgress AND NOT bCancelInProgress THEN
    bCancelInProgress := TRUE;
ELSE
	CancelMove := FALSE;
END_IF

IF bCancelInProgress THEN
    ProcessCancelOperation();
	
    RETURN; 
END_IF

(* 4. PROCESS NEW COMMAND *)
bisValidCmd := F_ValidateCommand(sInput := sRequestedActuator, nX => nX, sY => sY, sZ => sZ);
bisLinearActuator := sY = 'Chariot' OR sY = 'Compressor' OR sY = 'Sensor' OR sY = 'HeatExCoupola' OR sY = 'RegenCoupola'; 

bCanProcessCommand :=
    NOT bOperationInProgress AND
    (sRequestedActuator <> 'none') AND
    (sRequestedActuator <> 'close') AND
    (bSafetyOk OR IsResetCommand(sZ) OR bisLinearActuator) AND // LinearActuator don't have built-in or physical reset function
    NOT bCriticalAlarm;
	
IF bCanProcessCommand THEN
  
    IF NOT bisValidCmd THEN      
        sRequestedActuator := 'close';
        bAwaitingHMIClose := TRUE;
        tmrHMICloseSignal(IN := FALSE); 
		
        RETURN; 
    END_IF
    
	bOperationInProgress := TRUE;
    
	// Get command data
    LinearActuator := F_GetLinearCommandValue(nX, sY);
    LinearActuatorCmd := F_GetLinearCommandMember(nX, sY);
    LinearTable := F_GetStepperCommandValue(nX, sY);
    LinearTableCmd := F_GetStepperCommandMember(nX, sY);
	
	// Set command type
    bisLinearTableHomeCmd := sY = 'Home' AND LinearTableCmd^.bHoming;
	bisLinearTableSetHomeCmd := sY = 'SetHome' AND LinearTableCmd^.bHoming;
    bisLinearTableMoveCmd := sY = 'Motor';
    bisResetCmd := sZ = 'Reset';
END_IF

(* 5. EXECUTE COMMAND *)
IF bOperationInProgress AND NOT bCancelInProgress THEN
    IF bisLinearActuator THEN
        ProcessLinearActuator();
    ELSIF bisLinearTableHomeCmd OR bisLinearTableSetHomeCmd THEN
        ProcessLinearTable(bHome := TRUE);
    ELSIF bisLinearTableMoveCmd THEN
        ProcessLinearTable(bHome := FALSE);
    END_IF
	
END_IF

METHOD EvaluateSystemSafety : BOOL
EvaluateSystemSafety := TRUE;

FOR i := 1 TO 5 DO
    EvaluateSystemSafety := EvaluateSystemSafety AND gSystemAlarmStatus.aZoneStatus[i].bOkToRun;
END_FOR
END_METHOD

METHOD IsResetCommand : BOOL
VAR_INPUT
    sResetFlag : STRING;  
END_VAR
IF sResetFlag = 'Reset' THEN
    IsResetCommand := TRUE;
ELSE
	// Default behavior
    IsResetCommand := bSafetyOk;
END_IF
END_METHOD

METHOD ProcessCancelOperation
VAR
	nCancelResult   : INT := 0;
END_VAR
IF bisLinearActuator THEN
    LinearActuator^.Stop(State => LinearActuatorCmd^.nStatus); //Linear Actuator stop fails silently with motion timed out

ELSIF bisLinearTableHomeCmd OR bisLinearTableMoveCmd THEN
	IF LinearTable^.KeepAlive() THEN
		nCancelResult := LinearTable^.Stop();
	ELSE
		nCancelResult := -1;
	END_IF
	
    CASE nCancelResult OF
        1: // Success
            LinearTable^.GetPosition(fCurrentPosition => CurrentPosition);
            LinearTableCmd^.nPosition := CurrentPosition;
            
            IF bisLinearTableHomeCmd THEN
                LinearTableCmd^.bHomed := FALSE;
                LinearTableCmd^.bHoming := FALSE;
            END_IF;

		0: // Operation in progress
			RETURN;
			
       -1: // Failure
            IF bisLinearTableHomeCmd THEN
                LinearTableCmd^.bHomed := FALSE;
                LinearTableCmd^.bHoming := FALSE;
            ELSE
                LinearTableCmd^.nPosition := -1;
            END_IF;
    END_CASE;
END_IF;

LinearTable^.PowerDown();

//Request Pop-up close
sRequestedActuator := 'close';
bAwaitingHMIClose := TRUE;

//Cleanup
bOperationInProgress := FALSE; //Stop processing even if cancel fails
bCancelInProgress := FALSE;
CancelMove := FALSE;
END_METHOD

METHOD ProcessLinearActuator
VAR
	bisExtendCmd : BOOL;
END_VAR
// Get command value
bisExtendCmd := LinearActuatorCmd^.bCommand;

(* 1. RESET COMMAND CHECK *)
IF bisResetCmd THEN
    LinearActuator^.Reset(State => LinearActuatorCmd^.nStatus); // Instantaneous read of prox seonsors
	
	Result := 1;

	sRequestedActuator := 'close';
    bAwaitingHMIClose := TRUE;
	
	bOperationInProgress := FALSE;
    RETURN;
END_IF

(* 2. EXECUTE MOVEMENT COMMAND *)
IF bisExtendCmd THEN
    Result := LinearActuator^.Extend();
ELSE
    Result := LinearActuator^.Home();
END_IF

CASE Result OF
    1: // Success   
        IF bisExtendCmd THEN
            LinearActuatorCmd^.nStatus := 1;
        ELSE
            LinearActuatorCmd^.nStatus := 0;
        END_IF
        
        sRequestedActuator := 'close';
        bAwaitingHMIClose := TRUE;
    	
		bOperationInProgress := FALSE;
		
    0: // Continue
        // Operation in progress
        
   -1: // Failure
        bOperationInProgress := FALSE;
		
        LinearActuatorCmd^.nStatus := -1;
        
        sRequestedActuator := 'close';
        bAwaitingHMIClose := TRUE;
END_CASE
END_METHOD

METHOD ProcessLinearTable
VAR_INPUT
	bHome : BOOL;
END_VAR
VAR
	Error : BOOL;
	nCmdInt : INT;
	nFetchPosition : INT := 0;
END_VAR
(* 1. WAIT FOR STEPPER POWER-UP *)
IF LinearTable^.KeepAlive(Error => Error) THEN
	nFetchPosition := LinearTable^.GetPosition(fCurrentPosition => CurrentPosition);
	
	CASE nFetchPosition OF
		1: //Continue
		
		0: //Continue
			RETURN;
		
		-1: LinearTableCmd^.nPosition := -1;      
            Result := -1;                         
            LinearTable^.PowerDown();             
            bOperationInProgress := FALSE;
			
			sRequestedActuator := 'close';
			bAwaitingHMIClose := TRUE;
			tmrHMICloseSignal(IN := FALSE);
			
            RETURN;           
	END_CASE
	
ELSIF Error THEN
	Result := -1;
ELSE
	RETURN;
END_IF
	
(* 2. RESET COMMAND CHECK *)
IF bisResetCmd THEN
	LinearTable^.bHoldKeepAlive := TRUE;
	
	IF LinearTable^.KeepAlive() THEN
		Result := LinearTable^.Reset(TRUE);
	ELSE
		Result := -1;
	END_IF

    CASE Result OF
        1: // Success	
            LinearTableCmd^.nPosition := CurrentPosition;
            
            sRequestedActuator := 'close';
            bAwaitingHMIClose := TRUE;
            tmrHMICloseSignal(IN := FALSE); 
			
			LinearTable^.PowerDown();
			
			bOperationInProgress := FALSE;
            RETURN;
            
        0: // Operation in progress
			RETURN;
            
       -1: // Failure	
            LinearTableCmd^.nPosition := -1;
            
            sRequestedActuator := 'close';
            bAwaitingHMIClose := TRUE;
            tmrHMICloseSignal(IN := FALSE);
			
			LinearTable^.PowerDown();
			
			bOperationInProgress := FALSE;
            RETURN;
    END_CASE
END_IF

(* 3. EXECUTE MOVEMENT COMMAND *)
IF bHome THEN
	LinearTableCmd^.bHomed := FALSE;
	
	IF bisLinearTableHomeCmd THEN
		IF LinearTable^.KeepAlive() THEN
			Result := LinearTable^.Home(FALSE);
		ELSE
			Result := -1;
		END_IF
	ELSE
		IF LinearTable^.KeepAlive() THEN
			Result := LinearTable^.Home(TRUE); //Forced homing
		ELSE
			Result := -1;
		END_IF
	END_IF
	LinearTableCmd^.nPosition := CurrentPosition;
ELSE
	IF LinearTable^.KeepAlive() THEN	
			nCmdInt := LREAL_TO_INT(LinearTableCmd^.nCommand);
			CASE nCmdInt OF
				-1: Result := LinearTable^.Jog(Mode := MC_JOGMODE_STANDARD_SLOW, JogDir := TRUE, Execute := TRUE);
				
				-2: Result := LinearTable^.Jog(Mode := MC_JOGMODE_STANDARD_FAST, JogDir := TRUE, Execute := TRUE);
				
				-3: Result := LinearTable^.Jog(Mode := MC_JOGMODE_STANDARD_SLOW, JogDir := FALSE, Execute := TRUE);
				
				-4: Result := LinearTable^.Jog(Mode := MC_JOGMODE_STANDARD_FAST, JogDir := FALSE, Execute := TRUE);	

				-5: Result := LinearTable^.Jog(Execute := FALSE);	
			ELSE
				Result := LinearTable^.MoveToPosition(fPosition := LinearTableCmd^.nCommand, fVelocity := LinearTableCmd^.fVelocity);
			END_CASE		
			LinearTableCmd^.nPosition := CurrentPosition;
	ELSE
		Result := -1;
	END_IF
END_IF

CASE Result OF
    1: // Success
        IF bHome THEN    
            LinearTableCmd^.bHomed := TRUE;
            LinearTableCmd^.bHoming := FALSE;
        END_IF
        
		IF nCmdInt >= 0 THEN
			sRequestedActuator := 'close';
			bAwaitingHMIClose := TRUE;
			tmrHMICloseSignal(IN := FALSE);
		END_IF
		
		LinearTable^.PowerDown();
    	
		bOperationInProgress := FALSE;
		
    0: // Continue
        // Operation in progress
    
   -1: // Failure
        IF bHome THEN    
            LinearTableCmd^.bHomed := FALSE;
            LinearTableCmd^.bHoming := FALSE;
        ELSE
            LinearTableCmd^.nPosition := -1;
        END_IF
        
        IF nCmdInt >= 0 THEN
			sRequestedActuator := 'close';
			bAwaitingHMIClose := TRUE;
			tmrHMICloseSignal(IN := FALSE);
		END_IF
		
		LinearTable^.PowerDown();
		
		bOperationInProgress := FALSE;
END_CASE
END_METHOD

END_PROGRAM

// ---- POUs/FunctionBlocks/FB_LinearActuator.TcPOU
FUNCTION_BLOCK FB_LinearActuator
VAR
    // STATE & CONFIGURATION
    eState      : ENUM_LinearActuatorState := LAS_LinearActuator_Uninitialised;
    tTimeout    : TIME := T#30S;

    // ERROR HANDLING
    bError      : BOOL;
    sErrorMsg   : STRING(80);
	bHoldDriveFaulted : BOOL;
	fbDelayTimerHome : TON;
	fbDelayTimerExtend : TON;
	
    // REFERENCES
    pActuator   : POINTER TO ST_LinearActuator;

    // EDGE SELECTION FLAGS 
    bProxInRisingEdge   : BOOL := TRUE;   
    bProxOutRisingEdge  : BOOL := TRUE;  
    bProx2RisingEdge    : BOOL := TRUE;    
    bProx3RisingEdge    : BOOL := TRUE;  
    bFirstCycle : BOOL := TRUE;
	
    // EDGE DETECTION TRIGGERS
    r_trig_proxIn   : R_TRIG;             
    f_trig_proxIn   : F_TRIG;            
    r_trig_proxOut  : R_TRIG;            
    f_trig_proxOut  : F_TRIG;            
    r_trig_prox2    : R_TRIG;
    f_trig_prox2    : F_TRIG;
    r_trig_prox3    : R_TRIG;
    f_trig_prox3    : F_TRIG;
    
    // HELPER VARIABLES
    bIsGui   : BOOL;  
	bIsCmp   : BOOL;
    bIsBasic      : BOOL; 
	bIsPiv : BOOL; 
    bDetectError : BOOL;
	
    // EDGE DETECTION RESULTS
    bProxInDetected     : BOOL;
    bProxOutDetected    : BOOL;
    bProx2Detected      : BOOL;
    bProx3Detected      : BOOL;

END_VAR

METHOD CheckDriveFault : BOOL
VAR
	pAlarmCondition : POINTER TO BOOL;
END_VAR
IF NOT bIsBasic THEN
	pAlarmCondition := F_GetLinearActuatorAlarmCondition(pActuator^.sName, 'DriveFaulted');
	
    IF pActuator^.bFaultDI^ := TRUE THEN
		IF NOT bHoldDriveFaulted THEN
			eState := LAS_LinearActuator_Error;
		END_IF
		
		bHoldDriveFaulted := TRUE;
		IF pAlarmCondition <> 0 THEN
			pAlarmCondition^ := TRUE;
		END_IF
	ELSE
		IF pAlarmCondition <> 0 THEN
			pAlarmCondition^ := FALSE;
		END_IF
	END_IF
END_IF
END_METHOD

METHOD Extend : INT
VAR
    pAlarmCondition : POINTER TO BOOL;
	nStop : INT;
END_VAR
Extend := 0;

//CheckDriveFault();
UpdateProxDetection();

IF bFirstCycle AND NOT bIsPiv THEN
	GetPosition();
	bFirstCycle := FALSE;
END_IF

CASE eState OF
    LAS_LinearActuator_Retracted, LAS_LinearActuator_Error, LAS_LinearActuator_AtProx2, LAS_LinearActuator_AtProx3: //Allow Linear Actuator movement when position is unknown
		IF bIsGui THEN
			pActuator^.bStopControlDO^ := FALSE;
			pActuator^.bSpeedControlDO^ := FALSE;
		ELSIF bIsCmp THEN
			pActuator^.bStopControlDO^ := FALSE;
		END_IF
		
        SetForwardMovement();
		pActuator^.tTimeout(IN := TRUE, PT := tTimeout);
        eState := LAS_LinearActuator_Extending;

    LAS_LinearActuator_Extending:
		pActuator^.tTimeout(IN := TRUE, PT := tTimeout);
		
		IF bCriticalAlarm THEN
			pActuator^.tTimeout(IN := FALSE);
            Stop(); 
			//bHoldDriveFaulted := FALSE;
			
			IF bIsGui THEN
				pActuator^.bSpeedControlDO^ := FALSE;
			END_IF
			bFirstCycle := TRUE;
            Extend := -1;
		END_IF
		
		IF bIsBasic THEN
			SetForwardMovement(); //Continuous call of basic linear actuators
		END_IF
		
		IF bProx2Detected THEN
			IF bIsCmp THEN
				eState := LAS_LinearActuator_Error;		
				pAlarmCondition := F_GetLinearActuatorAlarmCondition(pActuator^.sName, 'UnknownPosition');
				IF pAlarmCondition <> 0 THEN
					pAlarmCondition^ := TRUE;
				END_IF
				
				Stop();
				
				IF bIsGui THEN
					pActuator^.bSpeedControlDO^ := FALSE;
				END_IF
				
				pActuator^.tTimeout(IN := FALSE);
				bHoldDriveFaulted := FALSE;
				bFirstCycle := TRUE;
				Extend := -1; 
			END_IF
		ELSIF bProx3Detected THEN
			IF pActuator^.bSpeedControlDO <> 0 THEN
				pActuator^.bSpeedControlDO^ := TRUE;  // Slow down when reaching Prox3
			END_IF
		END_IF
		
        IF bProxOutDetected THEN
			IF NOT bIsPiv THEN
				Stop();
			END_IF

			eState := LAS_LinearActuator_Extended;
			bHoldDriveFaulted := FALSE;
			bFirstCycle := TRUE;
		    pActuator^.tTimeout(IN := FALSE);
        END_IF
        
        IF pActuator^.tTimeout.Q THEN // Check for timeout
			Stop();
            eState := LAS_LinearActuator_Error;
            
            pAlarmCondition := F_GetLinearActuatorAlarmCondition(pActuator^.sName, 'MotionTimedOut');
            IF pAlarmCondition <> 0 THEN
                pAlarmCondition^ := TRUE;
            END_IF
            
			IF bIsGui THEN
				pActuator^.bSpeedControlDO^ := FALSE;
			END_IF
			
			pActuator^.tTimeout(IN := FALSE);
			bHoldDriveFaulted := FALSE;
			bFirstCycle := TRUE;
            Extend := -1;
        END_IF

    LAS_LinearActuator_Extended:		
		IF bIsPiv THEN
			fbDelayTimerExtend(IN := TRUE, PT := T#1S);		
			GetPosition();
			
			IF fbDelayTimerExtend.Q THEN
				Extend := 1; 
				Stop();
				bFirstCycle := TRUE;			
				fbDelayTimerExtend(IN := FALSE); 		
			END_IF		
		ELSE
			Extend := 1; 
			bFirstCycle := TRUE;
			
			IF bIsGui THEN
				pActuator^.bSpeedControlDO^ := FALSE;
			END_IF
		END_IF       
END_CASE
END_METHOD

METHOD FB_Init: BOOL
VAR_INPUT
    bInitRetains: BOOL;
    bInCopyCode: BOOL;   
    Actuator : POINTER TO ST_LinearActuator;  
END_VAR
VAR
    pAlarmCondition : POINTER TO BOOL;
END_VAR
pActuator := Actuator;
bHoldDriveFaulted := FALSE;

(* Detect actuator type *)
bIsGui := pActuator^.sName = 'HeatExCoupola3' OR pActuator^.sName = 'RegenCoupola3';
bIsCmp := pActuator^.sName = 'Compressor1' OR pActuator^.sName = 'Compressor3';
bIsPiv := pActuator^.sName = 'Sensor1';
bIsBasic := NOT bIsGui AND NOT bIsCmp;

(* Initialise speed control to fast *)
IF bIsGui THEN
    pActuator^.bSpeedControlDO^ := FALSE; 
END_IF

(* Initialise stop to false *)
IF NOT bIsBasic THEN
	pActuator^.bStopControlDO^ := FALSE; 
END_IF

IF bIsPiv THEN
	eState := LAS_LinearActuator_Retracted;
END_IF

//GetPosition();
END_METHOD

METHOD GetPosition : BOOL
VAR
	pAlarmCondition : POINTER TO BOOL;
END_VAR
VAR_OUTPUT
	State : SINT;
END_VAR
bDetectError := FALSE;
UpdateProxDetection();

IF bProxInRisingEdge = pActuator^.bProxIn^ THEN    
    eState := LAS_LinearActuator_Retracted;
    State := 0;  
	GetPosition := TRUE;
	bDetectError := TRUE;
END_IF

IF bIsCmp THEN
	IF bProxOutRisingEdge = (NOT pActuator^.bProxOut^) THEN //ProxOut is NC
    eState := LAS_LinearActuator_Extended;
    State := 1;  
	GetPosition := TRUE;
	bDetectError := TRUE;
	END_IF
ELSE
	IF bProxOutRisingEdge = pActuator^.bProxOut^ THEN
		eState := LAS_LinearActuator_Extended;
		State := 1;  
		GetPosition := TRUE;
		bDetectError := TRUE;
	END_IF
END_IF

IF bIsGui AND NOT bDetectError THEN
	IF bProx2RisingEdge = pActuator^.bProx2^ THEN
		eState := LAS_LinearActuator_AtProx2;
		State := 2;  
		GetPosition := TRUE;
		bDetectError := TRUE;
	ELSIF bProx3RisingEdge = pActuator^.bProx3^ THEN
		eState := LAS_LinearActuator_AtProx3;
		State := 3;  
		GetPosition := TRUE;
		bDetectError := TRUE;
	END_IF
END_IF

IF NOT bDetectError THEN
	eState := LAS_LinearActuator_Error;
	
	pAlarmCondition := F_GetLinearActuatorAlarmCondition(pActuator^.sName, 'UnknownPosition');
	IF pAlarmCondition <> 0 THEN
		pAlarmCondition^ := TRUE;
	END_IF

	State := -1;
	GetPosition := FALSE;
END_IF
END_METHOD

METHOD Home : INT
VAR
    pAlarmCondition : POINTER TO BOOL;
	nStop : INT;
	fbDelayTimer : TON;
END_VAR
Home := 0;

//CheckDriveFault();
UpdateProxDetection();

IF bFirstCycle AND NOT bIsPiv THEN
	GetPosition();
	bFirstCycle := FALSE;
END_IF

CASE eState OF
    LAS_LinearActuator_Extended, LAS_LinearActuator_Error, LAS_LinearActuator_AtProx2, LAS_LinearActuator_AtProx3: //Allow Linear Actuator movement when position is unknown
		IF bIsGui THEN
			pActuator^.bStopControlDO^ := FALSE;
			pActuator^.bSpeedControlDO^ := FALSE;
		ELSIF bIsCmp THEN
			pActuator^.bStopControlDO^ := FALSE;
		END_IF
		SetBackwardMovement();
		pActuator^.tTimeout(IN := TRUE, PT := tTimeout);
        eState := LAS_LinearActuator_Retracting;

    LAS_LinearActuator_Retracting:
		IF bCriticalAlarm THEN
			pActuator^.tTimeout(IN := FALSE);
            Stop(); 
			//bHoldDriveFaulted := FALSE;
			IF bIsGui THEN
				pActuator^.bSpeedControlDO^ := FALSE;
			END_IF
			bFirstCycle := TRUE;
            Home := -1;
		END_IF
		
		pActuator^.tTimeout(IN := TRUE, PT := tTimeout);
		
		IF bIsBasic THEN
			SetBackwardMovement(); //Continuous call of basic linear actuators
		END_IF
		
        IF bIsGui THEN
            IF bProx2Detected THEN
                IF pActuator^.bSpeedControlDO <> 0 THEN
                    pActuator^.bSpeedControlDO^ := TRUE;  // Slow down when reaching Prox2
                END_IF
            END_IF
        END_IF
        
        IF bProxInDetected THEN
			IF NOT bIsPiv THEN
				Stop();
			END_IF
			
			eState := LAS_LinearActuator_Retracted;
			bHoldDriveFaulted := FALSE;
			bFirstCycle := TRUE;
		    pActuator^.tTimeout(IN := FALSE);
        END_IF
        
        // Check for timeout
        IF pActuator^.tTimeout.Q THEN
			Stop(); 
            eState := LAS_LinearActuator_Error;
            pActuator^.tTimeout(IN := FALSE);
			
            pAlarmCondition := F_GetLinearActuatorAlarmCondition(pActuator^.sName, 'MotionTimedOut');
            IF pAlarmCondition <> 0 THEN
                pAlarmCondition^ := TRUE;
            END_IF
            
			IF bIsGui THEN
				pActuator^.bSpeedControlDO^ := FALSE;
			END_IF
			
            pActuator^.tTimeout(IN := FALSE);
			bHoldDriveFaulted := FALSE;
			bFirstCycle := TRUE;
            Home := -1;
        END_IF

    LAS_LinearActuator_Retracted:
		IF bIsPiv THEN
			fbDelayTimerHome(IN := TRUE, PT := T#1S);		
			GetPosition();
			
			IF fbDelayTimerHome.Q THEN
				Home := 1; 
				Stop();
				bFirstCycle := TRUE;			
				fbDelayTimerHome(IN := FALSE); 		
			END_IF		
		ELSE
			Home := 1; 
			bFirstCycle := TRUE;
			
			IF bIsGui THEN
				pActuator^.bSpeedControlDO^ := FALSE;
			END_IF
		END_IF       
END_CASE
END_METHOD

METHOD Reset : BOOL
VAR
    i : UINT;
    sActuatorName : STRING(50);
	pAlarmCondition : POINTER TO BOOL;
END_VAR
VAR_OUTPUT
    State : SINT;
END_VAR
sActuatorName := pActuator^.sName;

//CheckDriveFault();

IF NOT bIsPiv THEN
	IF GetPosition(State => State) THEN
		pAlarmCondition := F_GetLinearActuatorAlarmCondition(pActuator^.sName, 'UnknownPosition');
		IF pAlarmCondition <> 0 THEN
			pAlarmCondition^ := FALSE;
		END_IF
		
		pAlarmCondition := F_GetLinearActuatorAlarmCondition(pActuator^.sName, 'MotionTimedOut');
		IF pAlarmCondition <> 0 THEN
			pAlarmCondition^ := FALSE;
		END_IF
	END_IF
END_IF
END_METHOD

METHOD SetBackwardMovement : BOOL
VAR_INPUT
END_VAR
pActuator^.bFwdDO^ := FALSE;
pActuator^.bBckwDO^ := TRUE;
END_METHOD

METHOD SetForwardMovement : BOOL
pActuator^.bFwdDO^ := TRUE;
pActuator^.bBckwDO^ := FALSE;
END_METHOD

METHOD Stop : INT

VAR_OUTPUT
	State : SINT;
END_VAR
//CheckDriveFault();

pActuator^.bFwdDO^ := FALSE;
pActuator^.bBckwDO^ := FALSE;
pActuator^.tTimeout(IN := FALSE);

IF NOT bIsBasic THEN
	pActuator^.bStopControlDO^ := TRUE;
END_IF

GetPosition(State => State);
END_METHOD

METHOD UpdateProxDetection : BOOL
r_trig_proxIn(CLK := pActuator^.bProxIn^);
f_trig_proxIn(CLK := pActuator^.bProxIn^);

IF bIsCmp THEN
	r_trig_proxOut(CLK := (NOT pActuator^.bProxOut^));
	f_trig_proxOut(CLK := (NOT pActuator^.bProxOut^));
ELSE
	r_trig_proxOut(CLK := pActuator^.bProxOut^);
	f_trig_proxOut(CLK := pActuator^.bProxOut^);
END_IF

(* Select which edge is valid based on configuration flags *)
bProxInDetected := (bProxInRisingEdge AND r_trig_proxIn.Q) OR (NOT bProxInRisingEdge AND f_trig_proxIn.Q);
bProxOutDetected := (bProxOutRisingEdge AND r_trig_proxOut.Q) OR (NOT bProxOutRisingEdge AND f_trig_proxOut.Q);

IF NOT bIsBasic THEN
    r_trig_prox2(CLK := pActuator^.bProx2^);
    f_trig_prox2(CLK := pActuator^.bProx2^);
	
	bProx2Detected := (bProx2RisingEdge AND r_trig_prox2.Q) OR (NOT bProx2RisingEdge AND f_trig_prox2.Q);
	
	IF bIsGui THEN
		r_trig_prox3(CLK := pActuator^.bProx3^);
    	f_trig_prox3(CLK := pActuator^.bProx3^);
      
    	bProx3Detected := (bProx3RisingEdge AND r_trig_prox3.Q) OR (NOT bProx3RisingEdge AND f_trig_prox3.Q);
	END_IF
END_IF
END_METHOD

END_FUNCTION_BLOCK

// ---- POUs/Helper/F_GetLinearActuatorAlarmCondition.TcPOU
FUNCTION F_GetLinearActuatorAlarmCondition : POINTER TO BOOL
VAR_INPUT
    sActuatorName : STRING(50);    
    sAlarmType : STRING(50);      
END_VAR
VAR
    nRail : SINT;
    sBaseType : STRING(50);
    sLastChar : STRING(1);
    nNameLength : INT;
    pResult : POINTER TO BOOL;
END_VAR

// ============================================================================
// EXTRACT RAIL NUMBER FROM ACTUATOR NAME
// ============================================================================
nNameLength := LEN(sActuatorName);
IF nNameLength > 0 THEN
    sLastChar := RIGHT(sActuatorName, 1);
    nRail := STRING_TO_SINT(sLastChar);
    
    // Extract base type (everything except the last character)
    sBaseType := LEFT(sActuatorName, nNameLength - 1);
ELSE
    F_GetLinearActuatorAlarmCondition := 0;
    RETURN;
END_IF

// ============================================================================
// VALIDATE RAIL NUMBER
// ============================================================================
IF nRail < 1 OR nRail > 4 THEN
    F_GetLinearActuatorAlarmCondition := 0;
    RETURN;
END_IF

// ============================================================================
// MAP TO SPECIFIC ALARMS BASED ON RAIL, BASE TYPE, AND ALARM TYPE
// ============================================================================
IF nRail = 1 THEN
    // Rail 1 Alarms
    IF sBaseType = 'Sensor' THEN
        IF sAlarmType = 'MotionTimedOut' THEN
            pResult := ADR(GVL_Alarms.R1_Sensor_MotionTimedOut.bCondition);
        ELSIF sAlarmType = 'UnknownPosition' THEN
            pResult := ADR(GVL_Alarms.R1_Sensor_UnknownPosition.bCondition);
        END_IF
        
    ELSIF sBaseType = 'Compressor' THEN
        IF sAlarmType = 'MotionTimedOut' THEN
            pResult := ADR(GVL_Alarms.R1_Compressor_MotionTimedOut.bCondition);
        ELSIF sAlarmType = 'UnknownPosition' THEN
            pResult := ADR(GVL_Alarms.R1_Compressor_UnknownPosition.bCondition);
        END_IF
        
    ELSIF sBaseType = 'Chariot' THEN
        IF sAlarmType = 'MotionTimedOut' THEN
            pResult := ADR(GVL_Alarms.R1_Chariot_MotionTimedOut.bCondition);
        ELSIF sAlarmType = 'UnknownPosition' THEN
            pResult := ADR(GVL_Alarms.R1_Chariot_UnknownPosition.bCondition);
        END_IF
    END_IF
    
ELSIF nRail = 2 THEN
    // Rail 2 Alarms
    IF sBaseType = 'Chariot' THEN
        IF sAlarmType = 'MotionTimedOut' THEN
            pResult := ADR(GVL_Alarms.R2_Chariot_MotionTimedOut.bCondition);
        ELSIF sAlarmType = 'UnknownPosition' THEN
            pResult := ADR(GVL_Alarms.R2_Chariot_UnknownPosition.bCondition);
        END_IF
    END_IF
    
ELSIF nRail = 3 THEN
    // Rail 3 Alarms
    IF sBaseType = 'Compressor' THEN
        IF sAlarmType = 'MotionTimedOut' THEN
            pResult := ADR(GVL_Alarms.R3_Compressor_MotionTimedOut.bCondition);
        ELSIF sAlarmType = 'UnknownPosition' THEN
            pResult := ADR(GVL_Alarms.R3_Compressor_UnknownPosition.bCondition);
        END_IF
        
    ELSIF sBaseType = 'HeatExCoupola' THEN
        IF sAlarmType = 'MotionTimedOut' THEN
            pResult := ADR(GVL_Alarms.R3_HeatExCoupola_MotionTimedOut.bCondition);
        ELSIF sAlarmType = 'UnknownPosition' THEN
            pResult := ADR(GVL_Alarms.R3_HeatExCoupola_UnknownState.bCondition);
		ELSIF sAlarmType = 'DriveFaulted' THEN
			pResult := ADR(GVL_Alarms.R3_HeatExCoupola_DriveFaulted.bCondition);
        END_IF
        
    ELSIF sBaseType = 'RegenCoupola' THEN
        IF sAlarmType = 'MotionTimedOut' THEN
            pResult := ADR(GVL_Alarms.R3_RegenCoupola_MotionTimedOut.bCondition);
        ELSIF sAlarmType = 'UnknownPosition' THEN
            pResult := ADR(GVL_Alarms.R3_RegenCoupola_UnknownPosition.bCondition);
		ELSIF sAlarmType = 'DriveFaulted' THEN
			pResult := ADR(GVL_Alarms.R3_RegenCoupola_DriveFaulted.bCondition);
        END_IF
        
    ELSIF sBaseType = 'Chariot' THEN
        IF sAlarmType = 'MotionTimedOut' THEN
            pResult := ADR(GVL_Alarms.R3_Chariot_MotionTimedOut.bCondition);
        ELSIF sAlarmType = 'UnknownPosition' THEN
            pResult := ADR(GVL_Alarms.R3_Chariot_UnknownPosition.bCondition);
        END_IF
    END_IF
    
ELSIF nRail = 4 THEN
    // Rail 4 Alarms
    IF sBaseType = 'Chariot' THEN
        IF sAlarmType = 'MotionTimedOut' THEN
            pResult := ADR(GVL_Alarms.R4_Chariot_MotionTimedOut.bCondition);
        ELSIF sAlarmType = 'UnknownPosition' THEN
            pResult := ADR(GVL_Alarms.R4_Chariot_UnknownPosition.bCondition);
        END_IF
    END_IF
END_IF

F_GetLinearActuatorAlarmCondition := pResult;

END_FUNCTION

// ---- POUs/FunctionBlocks/FB_StepperMotor.TcPOU
FUNCTION_BLOCK FB_StepperMotor
VAR_INPUT
    nRail : SINT := 0; // Rail number / axis index
	bHoldKeepAlive : BOOL;
END_VAR

VAR
    // ==========================
    // Axis references & pointers
    // ==========================
    pAxis : POINTER TO AXIS_REF; // Pointer to axis reference
	pProx : POINTER TO BOOL;
	pRefPos : POINTER TO LREAL;
	pHomingOptions : POINTER TO ST_HomingOptions;

    // ======================
    // Motion control function blocks
    // ======================
    fbPower   : MC_Power;            // Power on/off control
    fbStop    : MC_Halt;             // Stop motion
    fbMoveAbs : MC_MoveAbsolute;     // Absolute move command
    fbHome    : MC_Home;             // Homing procedure
    fbRead    : MC_ReadActualPosition; // Read position
    fbReset   : MC_Reset;            // Reset errors
	fbReadError : MC_ReadAxisError;
	fbJog     : MC_Jog;

    // =================
    // Error & state handling
    // =================
    nErrID : UDINT; // Error ID
	
    eState : ENUM_StepperMotorState := LAS_Stepper_Idle; // Current state
	bIsUp : BOOL := FALSE;
	
    // ==========================
    // Hardware check variables
    // ==========================
    eHardwareCheckState   : ENUM_HardwareCheckState; // Hardware check state
END_VAR

METHOD FB_Init: BOOL
VAR_INPUT
    bInitRetains: BOOL; 
    bInCopyCode: BOOL;  
	
	init_axis : POINTER TO AXIS_REF;
	init_prox : POINTER TO BOOL;
	init_refpos : POINTER TO LREAL;
	init_homingoptions : POINTER TO ST_HomingOptions;
END_VAR
pAxis := init_axis;
pProx := init_prox;
pRefPos := init_refpos;
pHomingOptions := init_homingoptions;
END_METHOD

METHOD GetPosition : INT
VAR
	pAlarmCondition : POINTER TO BOOL;
	sErrorMsg : STRING(255);
END_VAR

VAR_OUTPUT
	fCurrentPosition : LREAL;
END_VAR
GetPosition := 0;

fbRead(Axis := pAxis^, Enable := TRUE, Position => fCurrentPosition);

IF fbRead.Busy THEN
	IF fbRead.Error THEN
		pAlarmCondition := F_GetStepperAlarmCondition(nRail, 'UnableToReadPosition');
		IF pAlarmCondition <> 0 THEN
			pAlarmCondition^ := TRUE;
		END_IF
		
		GetPosition := -1;
		sErrorMsg := F_GetMC2ErrorDescription(fbRead.ErrorID);
					
		CASE nRail OF
			1: GVL_Alarms.R1_Stepper_Motion_Failed.sMessage := CONCAT('Stepper rail 1 position read failed: ', sErrorMsg);
			2: GVL_Alarms.R2_Stepper_Motion_Failed.sMessage := CONCAT('Stepper rail 2 position read failed: ', sErrorMsg);
			3: GVL_Alarms.R3_Stepper_Motion_Failed.sMessage := CONCAT('Stepper rail 3 position read failed: ', sErrorMsg);
			4: GVL_Alarms.R4_Stepper_Motion_Failed.sMessage := CONCAT('Stepper rail 4 position read failed: ', sErrorMsg);
		END_CASE
	ELSIF fbRead.Valid THEN
		GetPosition := 1;
	ELSIF NOT fbRead.Valid THEN
	GetPosition := -1;
	END_IF
END_IF
END_METHOD

METHOD Home : INT
VAR_INPUT
	bIsForced : BOOL;    
END_VAR
VAR
    pAlarmCondition : POINTER TO BOOL; // Pointer to external alarm condition
	sErrorMsg : STRING(255);
END_VAR
Home := 0;

CASE eState OF
    LAS_Stepper_Ready, LAS_Stepper_Hardware_Check:
        IF bIsForced THEN
            fbHome(Axis := pAxis^, Execute := TRUE, HomingMode := MC_Direct, Position := pRefPos^);
            eState := LAS_Stepper_Homing;
		
		ELSE
			fbHome(Axis := pAxis^, Execute := TRUE, HomingMode := MC_DefaultHoming, Position := pRefPos^, bCalibrationCam := pProx^, Options := pHomingOptions^);
            eState := LAS_Stepper_Homing;
        END_IF
		
    LAS_Stepper_Homing:
		IF bIsForced THEN
			fbHome(Axis := pAxis^, Execute := TRUE, HomingMode := MC_Direct, Position := pRefPos^);
		ELSE
			fbHome(Axis := pAxis^, Execute := TRUE, HomingMode := MC_DefaultHoming, Position := pRefPos^, bCalibrationCam := pProx^, Options := pHomingOptions^);
		END_IF
        
        IF fbHome.Error THEN		
            eState := LAS_Stepper_Error;
            nErrID := fbHome.ErrorID;
			
			pAlarmCondition := F_GetStepperAlarmCondition(nRail, 'Homing_Failed');
            IF pAlarmCondition <> 0 THEN
                pAlarmCondition^ := TRUE;
                
                sErrorMsg := F_GetMC2ErrorDescription(fbHome.ErrorID);
                
                CASE nRail OF
                    1: GVL_Alarms.R1_Stepper_Homing_Failed.sMessage := CONCAT('Stepper rail 1 homing failed: ', sErrorMsg);
                    2: GVL_Alarms.R2_Stepper_Homing_Failed.sMessage := CONCAT('Stepper rail 2 homing failed: ', sErrorMsg);
                    3: GVL_Alarms.R3_Stepper_Homing_Failed.sMessage := CONCAT('Stepper rail 3 homing failed: ', sErrorMsg);
                    4: GVL_Alarms.R4_Stepper_Homing_Failed.sMessage := CONCAT('Stepper rail 4 homing failed: ', sErrorMsg);
                END_CASE
            END_IF
            
            Home := -1;

        ELSIF fbHome.Done THEN
            fbHome(Axis := pAxis^, Execute := FALSE);
			Home := 1; 
        END_IF
    
    LAS_Stepper_Error:
        Home := -1;
        
END_CASE
END_METHOD

METHOD Jog : INT
VAR_INPUT
	Mode : E_JOGMODE := MC_JOGMODE_STANDARD_SLOW; //Slow or Fast
	JogDir  : BOOL := TRUE;
	Execute : BOOL;
END_VAR

VAR
	pAlarmCondition : POINTER TO BOOL;
	sErrorMsg : STRING(255);
END_VAR
Jog := 0;

CASE eState OF
	LAS_Stepper_Ready, LAS_Stepper_Idle:
		IF Execute THEN
			fbJog(Axis := pAxis^, Mode := Mode, JogForward := JogDir, JogBackwards := NOT JogDir);
		END_IF
		eState := LAS_Stepper_Moving;

	LAS_Stepper_Moving:
		IF fbJog.Busy AND Execute THEN
			fbJog(Axis := pAxis^);
		ELSE
			fbJog(Axis := pAxis^, JogForward := FALSE, JogBackwards := FALSE);
		END_IF
		
		IF fbJog.Error THEN
			eState := LAS_Stepper_Error;
			nErrID := fbJog.ErrorID;
			
			pAlarmCondition := F_GetStepperAlarmCondition(nRail, 'Motion_Failed');
			IF pAlarmCondition <> 0 THEN
				pAlarmCondition^ := TRUE;
				
				sErrorMsg := F_GetMC2ErrorDescription(fbJog.ErrorID);
				
				CASE nRail OF
					1: GVL_Alarms.R1_Stepper_Motion_Failed.sMessage := CONCAT('Stepper rail 1 motion failed: ', sErrorMsg);
					2: GVL_Alarms.R2_Stepper_Motion_Failed.sMessage := CONCAT('Stepper rail 2 motion failed: ', sErrorMsg);
					3: GVL_Alarms.R3_Stepper_Motion_Failed.sMessage := CONCAT('Stepper rail 3 motion failed: ', sErrorMsg);
					4: GVL_Alarms.R4_Stepper_Motion_Failed.sMessage := CONCAT('Stepper rail 4 motion failed: ', sErrorMsg);
				END_CASE
			END_IF
			
			fbJog(Axis := pAxis^, JogForward := FALSE, JogBackwards := FALSE);
			Jog := -1;
		END_IF
				
		IF fbJog.Done THEN
			eState := LAS_Stepper_Ready;
			Jog := 1; 
			nErrID := 0;
		END_IF
	
	LAS_Stepper_Error:
		Jog := -1; 	
END_CASE
END_METHOD

METHOD KeepAlive : BOOL
VAR
	pAlarmCondition : POINTER TO BOOL;
	sErrorMsg : STRING(255);
END_VAR
VAR_OUTPUT
	Error : BOOL;
END_VAR
Error := FALSE;

IF NOT bHoldKeepAlive THEN
	fbPower(Axis := pAxis^, Enable := TRUE, Enable_positive := TRUE, Enable_Negative := TRUE, Override := 100);
	
	IF fbPower.Error THEN    
		eState := LAS_Stepper_PowerError;
		bIsUp := FALSE;
		
		pAlarmCondition := F_GetStepperAlarmCondition(nRail, 'PowerUp_Failed');
	   IF pAlarmCondition <> 0 THEN
			pAlarmCondition^ := TRUE;
	
			sErrorMsg := F_GetMC2ErrorDescription(fbPower.ErrorID);
			
			CASE nRail OF
				1: GVL_Alarms.R1_Stepper_PowerUp_Failed.sMessage :=  CONCAT('Stepper rail 1 powerup failed: ', sErrorMsg);
				2: GVL_Alarms.R2_Stepper_PowerUp_Failed.sMessage :=  CONCAT('Stepper rail 2 powerup failed: ', sErrorMsg);
				3: GVL_Alarms.R3_Stepper_PowerUp_Failed.sMessage :=  CONCAT('Stepper rail 3 powerup failed: ', sErrorMsg);
				4: GVL_Alarms.R4_Stepper_PowerUp_Failed.sMessage :=  CONCAT('Stepper rail 4 powerup failed: ', sErrorMsg);
			END_CASE
		END_IF
		
		Error := TRUE;
		KeepAlive := FALSE;
		
	ELSIF fbPower.Status THEN
		IF NOT bIsUp THEN
			bIsUp := TRUE;
			
			pAlarmCondition := F_GetStepperAlarmCondition(nRail, 'PowerUp_Failed');
			IF pAlarmCondition <> 0 THEN 
				pAlarmCondition^ := FALSE; 
			END_IF
			
			CASE nRail OF
				1: GVL_Alarms.R1_Stepper_PowerUp_Failed.sMessage := '';
				2: GVL_Alarms.R2_Stepper_PowerUp_Failed.sMessage := '';
				3: GVL_Alarms.R3_Stepper_PowerUp_Failed.sMessage := '';
				4: GVL_Alarms.R4_Stepper_PowerUp_Failed.sMessage := '';
			END_CASE
			
			CASE eState OF
				LAS_Stepper_PowerError:
					eState := LAS_Stepper_Error;
					
				LAS_Stepper_Error:
					// Keep State 
				
				LAS_Stepper_Idle:
					eState := LAS_Stepper_Ready;
			END_CASE
		END_IF
		
		KeepAlive := TRUE;
		
	ELSE
		// Power-up in progress
		KeepAlive := FALSE;
	END_IF
ELSE
	KeepAlive := TRUE;
END_IF
END_METHOD

METHOD MoveToPosition : INT
VAR_INPUT
    fPosition : LREAL;  // Target position
	fVelocity : LREAL;
END_VAR

VAR
	pAlarmCondition : POINTER TO BOOL;
	sErrorMsg : STRING(255);
END_VAR
MoveToPosition := 0;

CASE eState OF
	LAS_Stepper_Ready, LAS_Stepper_Idle:
		fbMoveAbs(Axis := pAxis^, Execute := TRUE, Position := fPosition, Velocity := fVelocity);
		eState := LAS_Stepper_Moving;

	LAS_Stepper_Moving:
		IF fbMoveAbs.Busy THEN
			fbMoveAbs(Axis := pAxis^);
		END_IF
		
		IF fbMoveAbs.Error THEN
			eState := LAS_Stepper_Error;
			nErrID := fbMoveAbs.ErrorID;
			
			pAlarmCondition := F_GetStepperAlarmCondition(nRail, 'Motion_Failed');
			IF pAlarmCondition <> 0 THEN
				pAlarmCondition^ := TRUE;
				
				sErrorMsg := F_GetMC2ErrorDescription(fbMoveAbs.ErrorID);
				
